  PROC DrawPart198()
    MoveL Offs(pOrigin,350.48,95.40,0.00),v40,z0,tPen\WObj:=wPaper;
    MoveL Offs(pOrigin,348.08,93.00,0.00),v40,z0,tPen\WObj:=wPaper;
    MoveL Offs(pOrigin,348.60,93.14,0.00),v40,z0,tPen\WObj:=wPaper;
    MoveL Offs(pOrigin,351.36,93.14,0.00),v40,z0,tPen\WObj:=wPaper;
    MoveL Offs(pOrigin,351.36,92.97,0.00),v40,z0,tPen\WObj:=wPaper;
    MoveL Offs(pOrigin,350.94,93.61,0.00),v40,z0,tPen\WObj:=wPaper;
    MoveL Offs(pOrigin,351.36,92.97,0.00),v40,z0,tPen\WObj:=wPaper;
    MoveL Offs(pOrigin,350.61,93.40,0.00),v40,z0,tPen\WObj:=wPaper;
    MoveL Offs(pOrigin,350.61,90.42,0.00),v40,z0,tPen\WObj:=wPaper;
    MoveL Offs(pOrigin,350.30,90.64,0.00),v40,z0,tPen\WObj:=wPaper;
    MoveL Offs(pOrigin,348.60,77.25,0.00),v40,z0,tPen\WObj:=wPaper;
    MoveL Offs(pOrigin,348.81,76.82,0.00),v40,z0,tPen\WObj:=wPaper;
    MoveL Offs(pOrigin,351.36,77.04,0.00),v40,z0,tPen\WObj:=wPaper;
    MoveL Offs(pOrigin,352.42,77.46,0.00),v40,z0,tPen\WObj:=wPaper;
    MoveL Offs(pOrigin,351.79,82.35,0.00),v40,z0,tPen\WObj:=wPaper;
    MoveL Offs(pOrigin,351.58,87.66,0.00),v40,z0,tPen\WObj:=wPaper;
    MoveL Offs(pOrigin,350.94,90.21,0.00),v40,z0,tPen\WObj:=wPaper;
    MoveL Offs(pOrigin,350.30,91.28,0.00),v40,fine,tPen\WObj:=wPaper;
    MoveL Offs(pOrigin,350.30,91.28,6.00),v60,z5,tPen\WObj:=wPaper;
    MoveL Offs(pOrigin,348.07,90.00,6.00),vTravel,z5,tPen\WObj:=wPaper;
    MoveL Offs(pOrigin,348.07,90.00,0.00),v60,z0,tPen\WObj:=wPaper;
    MoveL Offs(pOrigin,351.83,93.76,0.00),v40,z0,tPen\WObj:=wPaper;
    MoveL Offs(pOrigin,350.73,93.82,0.00),v40,z0,tPen\WObj:=wPaper;
    MoveL Offs(pOrigin,350.30,94.46,0.00),v40,z0,tPen\WObj:=wPaper;
    MoveL Offs(pOrigin,350.73,93.82,0.00),v40,fine,tPen\WObj:=wPaper;
    MoveL Offs(pOrigin,350.73,93.82,6.00),v60,z5,tPen\WObj:=wPaper;
    MoveL Offs(pOrigin,347.54,90.28,6.00),vTravel,z5,tPen\WObj:=wPaper;
    MoveL Offs(pOrigin,347.54,90.28,0.00),v60,z0,tPen\WObj:=wPaper;
    MoveL Offs(pOrigin,354.30,83.51,0.00),v40,z0,tPen\WObj:=wPaper;
    MoveL Offs(pOrigin,353.89,83.88,0.00),v40,z0,tPen\WObj:=wPaper;
    MoveL Offs(pOrigin,351.49,81.47,0.00),v40,z0,tPen\WObj:=wPaper;
    MoveL Offs(pOrigin,352.00,81.53,0.00),v40,z0,tPen\WObj:=wPaper;
    MoveL Offs(pOrigin,353.49,81.53,0.00),v40,z0,tPen\WObj:=wPaper;
    MoveL Offs(pOrigin,354.03,81.03,0.00),v40,z0,tPen\WObj:=wPaper;
    MoveL Offs(pOrigin,351.63,78.63,0.00),v40,z0,tPen\WObj:=wPaper;
    MoveL Offs(pOrigin,352.21,78.36,0.00),v40,z0,tPen\WObj:=wPaper;
    MoveL Offs(pOrigin,354.12,78.36,0.00),v40,z0,tPen\WObj:=wPaper;
    MoveL Offs(pOrigin,353.77,77.89,0.00),v40,z0,tPen\WObj:=wPaper;
    MoveL Offs(pOrigin,353.77,76.40,0.00),v40,fine,tPen\WObj:=wPaper;
    MoveL Offs(pOrigin,353.77,76.40,6.00),v60,z5,tPen\WObj:=wPaper;
    MoveL Offs(pOrigin,352.53,74.83,6.00),vTravel,z5,tPen\WObj:=wPaper;
    MoveL Offs(pOrigin,352.53,74.83,0.00),v60,z0,tPen\WObj:=wPaper;
    MoveL Offs(pOrigin,346.52,80.84,0.00),v40,fine,tPen\WObj:=wPaper;
    MoveL Offs(pOrigin,346.52,80.84,6.00),v60,z5,tPen\WObj:=wPaper;
    MoveL Offs(pOrigin,346.38,79.49,6.00),vTravel,z5,tPen\WObj:=wPaper;
    MoveL Offs(pOrigin,346.38,79.49,0.00),v60,z0,tPen\WObj:=wPaper;
    MoveL Offs(pOrigin,351.34,74.54,0.00),v40,z0,tPen\WObj:=wPaper;
    MoveL Offs(pOrigin,351.17,75.18,0.00),v40,z0,tPen\WObj:=wPaper;
    MoveL Offs(pOrigin,354.93,78.94,0.00),v40,fine,tPen\WObj:=wPaper;
    MoveL Offs(pOrigin,354.93,78.94,6.00),v60,z5,tPen\WObj:=wPaper;
    MoveL Offs(pOrigin,355.66,80.66,6.00),vTravel,z5,tPen\WObj:=wPaper;
    MoveL Offs(pOrigin,355.66,80.66,0.00),v60,z0,tPen\WObj:=wPaper;
    MoveL Offs(pOrigin,361.07,75.25,0.00),v40,z0,tPen\WObj:=wPaper;
    MoveL Offs(pOrigin,360.76,75.81,0.00),v40,z0,tPen\WObj:=wPaper;
    MoveL Offs(pOrigin,368.57,83.62,0.00),v40,z0,tPen\WObj:=wPaper;
    MoveL Offs(pOrigin,368.83,83.92,0.00),v40,z0,tPen\WObj:=wPaper;
    MoveL Offs(pOrigin,373.49,79.26,0.00),v40,z0,tPen\WObj:=wPaper;
    MoveL Offs(pOrigin,373.65,79.75,0.00),v40,z0,tPen\WObj:=wPaper;
    MoveL Offs(pOrigin,374.86,80.95,0.00),v40,fine,tPen\WObj:=wPaper;
    MoveL Offs(pOrigin,374.86,80.95,6.00),v60,z5,tPen\WObj:=wPaper;
    MoveL Offs(pOrigin,373.36,80.94,6.00),vTravel,z5,tPen\WObj:=wPaper;
    MoveL Offs(pOrigin,373.36,80.94,0.00),v60,z0,tPen\WObj:=wPaper;
    MoveL Offs(pOrigin,372.46,80.04,0.00),v40,z0,tPen\WObj:=wPaper;
    MoveL Offs(pOrigin,371.99,79.27,0.00),v40,z0,tPen\WObj:=wPaper;
    MoveL Offs(pOrigin,367.79,83.47,0.00),v40,z0,tPen\WObj:=wPaper;
    MoveL Offs(pOrigin,366.89,82.88,0.00),v40,z0,tPen\WObj:=wPaper;
    MoveL Offs(pOrigin,370.49,79.27,0.00),v40,z0,tPen\WObj:=wPaper;
    MoveL Offs(pOrigin,370.96,80.04,0.00),v40,z0,tPen\WObj:=wPaper;
    MoveL Offs(pOrigin,371.86,80.94,0.00),v40,fine,tPen\WObj:=wPaper;
    MoveL Offs(pOrigin,371.86,80.94,6.00),v60,z5,tPen\WObj:=wPaper;
    MoveL Offs(pOrigin,372.40,82.58,6.00),vTravel,z5,tPen\WObj:=wPaper;
    MoveL Offs(pOrigin,372.40,82.58,0.00),v60,z0,tPen\WObj:=wPaper;
    MoveL Offs(pOrigin,368.58,82.58,0.00),v40,fine,tPen\WObj:=wPaper;
    MoveL Offs(pOrigin,368.58,82.58,6.00),v60,z5,tPen\WObj:=wPaper;
    MoveL Offs(pOrigin,370.06,81.53,6.00),vTravel,z5,tPen\WObj:=wPaper;
    MoveL Offs(pOrigin,370.06,81.53,0.00),v60,z0,tPen\WObj:=wPaper;
    MoveL Offs(pOrigin,366.45,81.53,0.00),v40,fine,tPen\WObj:=wPaper;
    MoveL Offs(pOrigin,366.45,81.53,6.00),v60,z5,tPen\WObj:=wPaper;
    MoveL Offs(pOrigin,364.94,81.83,6.00),vTravel,z5,tPen\WObj:=wPaper;
    MoveL Offs(pOrigin,364.94,81.83,0.00),v60,z0,tPen\WObj:=wPaper;
    MoveL Offs(pOrigin,367.80,78.98,0.00),v40,fine,tPen\WObj:=wPaper;
    MoveL Offs(pOrigin,367.80,78.98,6.00),v60,z5,tPen\WObj:=wPaper;
    MoveL Offs(pOrigin,368.36,80.47,6.00),vTravel,z5,tPen\WObj:=wPaper;
    MoveL Offs(pOrigin,368.36,80.47,0.00),v60,z0,tPen\WObj:=wPaper;
    MoveL Offs(pOrigin,364.54,80.47,0.00),v40,fine,tPen\WObj:=wPaper;
    MoveL Offs(pOrigin,364.54,80.47,6.00),v60,z5,tPen\WObj:=wPaper;
    MoveL Offs(pOrigin,366.24,79.42,6.00),vTravel,z5,tPen\WObj:=wPaper;
    MoveL Offs(pOrigin,366.24,79.42,0.00),v60,z0,tPen\WObj:=wPaper;
    MoveL Offs(pOrigin,362.84,79.42,0.00),v40,z0,tPen\WObj:=wPaper;
    MoveL Offs(pOrigin,362.22,78.74,0.00),v40,z0,tPen\WObj:=wPaper;
    MoveL Offs(pOrigin,362.22,77.04,0.00),v40,z0,tPen\WObj:=wPaper;
    MoveL Offs(pOrigin,361.17,76.82,0.00),v40,z0,tPen\WObj:=wPaper;
    MoveL Offs(pOrigin,361.17,78.31,0.00),v40,fine,tPen\WObj:=wPaper;
    MoveL Offs(pOrigin,361.17,78.31,6.00),v60,z5,tPen\WObj:=wPaper;
    MoveL Offs(pOrigin,359.11,78.71,6.00),vTravel,z5,tPen\WObj:=wPaper;
    MoveL Offs(pOrigin,359.11,78.71,0.00),v60,z0,tPen\WObj:=wPaper;
    MoveL Offs(pOrigin,362.42,75.40,0.00),v40,fine,tPen\WObj:=wPaper;
    MoveL Offs(pOrigin,362.42,75.40,6.00),v60,z5,tPen\WObj:=wPaper;
    MoveL Offs(pOrigin,360.14,69.22,6.00),vTravel,z5,tPen\WObj:=wPaper;
    MoveL Offs(pOrigin,360.14,69.22,0.00),v60,z0,tPen\WObj:=wPaper;
    MoveL Offs(pOrigin,359.24,68.32,0.00),v40,fine,tPen\WObj:=wPaper;
    MoveL Offs(pOrigin,359.24,68.32,6.00),v60,z5,tPen\WObj:=wPaper;
    MoveL Offs(pOrigin,361.33,67.42,6.00),vTravel,z5,tPen\WObj:=wPaper;
    MoveL Offs(pOrigin,361.33,67.42,0.00),v60,z0,tPen\WObj:=wPaper;
    MoveL Offs(pOrigin,362.23,68.33,0.00),v40,z0,tPen\WObj:=wPaper;
    MoveL Offs(pOrigin,363.28,67.88,0.00),v40,z0,tPen\WObj:=wPaper;
    MoveL Offs(pOrigin,362.38,66.98,0.00),v40,fine,tPen\WObj:=wPaper;
    MoveL Offs(pOrigin,362.38,66.98,6.00),v60,z5,tPen\WObj:=wPaper;
    MoveL Offs(pOrigin,364.32,65.94,6.00),vTravel,z5,tPen\WObj:=wPaper;
    MoveL Offs(pOrigin,364.32,65.94,0.00),v60,z0,tPen\WObj:=wPaper;
    MoveL Offs(pOrigin,365.23,66.84,0.00),v40,z0,tPen\WObj:=wPaper;
    MoveL Offs(pOrigin,366.27,66.39,0.00),v40,z0,tPen\WObj:=wPaper;
    MoveL Offs(pOrigin,365.37,65.49,0.00),v40,fine,tPen\WObj:=wPaper;
    MoveL Offs(pOrigin,365.37,65.49,6.00),v60,z5,tPen\WObj:=wPaper;
    MoveL Offs(pOrigin,371.09,75.69,6.00),vTravel,z5,tPen\WObj:=wPaper;
    MoveL Offs(pOrigin,371.09,75.69,0.00),v60,z0,tPen\WObj:=wPaper;
    MoveL Offs(pOrigin,371.85,76.44,0.00),v40,fine,tPen\WObj:=wPaper;
    MoveL Offs(pOrigin,371.85,76.44,6.00),v60,z5,tPen\WObj:=wPaper;
    MoveL Offs(pOrigin,377.37,82.84,6.00),vTravel,z5,tPen\WObj:=wPaper;
    MoveL Offs(pOrigin,377.37,82.84,0.00),v60,z0,tPen\WObj:=wPaper;
  ENDPROC

  PROC DrawPart199()
    MoveL Offs(pOrigin,374.52,85.70,0.00),v40,fine,tPen\WObj:=wPaper;
    MoveL Offs(pOrigin,374.52,85.70,6.00),v60,z5,tPen\WObj:=wPaper;
    MoveL Offs(pOrigin,370.74,95.45,6.00),vTravel,z5,tPen\WObj:=wPaper;
    MoveL Offs(pOrigin,370.74,95.45,0.00),v60,z0,tPen\WObj:=wPaper;
    MoveL Offs(pOrigin,369.39,96.80,0.00),v40,z0,tPen\WObj:=wPaper;
    MoveL Offs(pOrigin,368.35,96.35,0.00),v40,z0,tPen\WObj:=wPaper;
    MoveL Offs(pOrigin,369.70,95.00,0.00),v40,z0,tPen\WObj:=wPaper;
    MoveL Offs(pOrigin,368.65,94.56,0.00),v40,z0,tPen\WObj:=wPaper;
    MoveL Offs(pOrigin,367.30,95.91,0.00),v40,fine,tPen\WObj:=wPaper;
    MoveL Offs(pOrigin,367.30,95.91,6.00),v60,z5,tPen\WObj:=wPaper;
    MoveL Offs(pOrigin,370.44,97.25,6.00),vTravel,z5,tPen\WObj:=wPaper;
    MoveL Offs(pOrigin,370.44,97.25,0.00),v60,z0,tPen\WObj:=wPaper;
    MoveL Offs(pOrigin,371.79,95.89,0.00),v40,z0,tPen\WObj:=wPaper;
    MoveL Offs(pOrigin,372.84,96.34,0.00),v40,z0,tPen\WObj:=wPaper;
    MoveL Offs(pOrigin,371.79,97.39,0.00),v40,fine,tPen\WObj:=wPaper;
    MoveL Offs(pOrigin,371.79,97.39,6.00),v60,z5,tPen\WObj:=wPaper;
    MoveL Offs(pOrigin,373.14,97.54,6.00),vTravel,z5,tPen\WObj:=wPaper;
    MoveL Offs(pOrigin,373.14,97.54,0.00),v60,z0,tPen\WObj:=wPaper;
    MoveL Offs(pOrigin,373.89,96.79,0.00),v40,fine,tPen\WObj:=wPaper;
    MoveL Offs(pOrigin,373.89,96.79,6.00),v60,z5,tPen\WObj:=wPaper;
    MoveL Offs(pOrigin,376.01,97.86,6.00),vTravel,z5,tPen\WObj:=wPaper;
    MoveL Offs(pOrigin,376.01,97.86,0.00),v60,z0,tPen\WObj:=wPaper;
    MoveL Offs(pOrigin,369.21,95.88,0.00),v40,z0,tPen\WObj:=wPaper;
    MoveL Offs(pOrigin,364.75,93.40,0.00),v40,z0,tPen\WObj:=wPaper;
    MoveL Offs(pOrigin,360.08,89.15,0.00),v40,z0,tPen\WObj:=wPaper;
    MoveL Offs(pOrigin,357.10,84.90,0.00),v40,fine,tPen\WObj:=wPaper;
    MoveL Offs(pOrigin,357.10,84.90,6.00),v60,z5,tPen\WObj:=wPaper;
    MoveL Offs(pOrigin,353.99,86.81,6.00),vTravel,z5,tPen\WObj:=wPaper;
    MoveL Offs(pOrigin,353.99,86.81,0.00),v60,z0,tPen\WObj:=wPaper;
    MoveL Offs(pOrigin,342.72,98.08,0.00),v40,fine,tPen\WObj:=wPaper;
    MoveL Offs(pOrigin,342.72,98.08,6.00),v60,z5,tPen\WObj:=wPaper;
    MoveL Offs(pOrigin,343.60,98.98,6.00),vTravel,z5,tPen\WObj:=wPaper;
    MoveL Offs(pOrigin,343.60,98.98,0.00),v60,z0,tPen\WObj:=wPaper;
    MoveL Offs(pOrigin,352.17,107.54,0.00),v40,z0,tPen\WObj:=wPaper;
    MoveL Offs(pOrigin,351.79,107.85,0.00),v40,z0,tPen\WObj:=wPaper;
    MoveL Offs(pOrigin,353.27,109.34,0.00),v40,z0,tPen\WObj:=wPaper;
    MoveL Offs(pOrigin,351.79,107.85,0.00),v40,fine,tPen\WObj:=wPaper;
    MoveL Offs(pOrigin,351.79,107.85,6.00),v60,z5,tPen\WObj:=wPaper;
    MoveL Offs(pOrigin,355.87,108.83,6.00),vTravel,z5,tPen\WObj:=wPaper;
    MoveL Offs(pOrigin,355.87,108.83,0.00),v60,z0,tPen\WObj:=wPaper;
    MoveL Offs(pOrigin,357.83,106.87,0.00),v40,z0,tPen\WObj:=wPaper;
    MoveL Offs(pOrigin,358.72,107.47,0.00),v40,z0,tPen\WObj:=wPaper;
    MoveL Offs(pOrigin,356.62,109.57,0.00),v40,z0,tPen\WObj:=wPaper;
    MoveL Offs(pOrigin,356.37,108.75,0.00),v40,z0,tPen\WObj:=wPaper;
    MoveL Offs(pOrigin,341.94,94.33,0.00),v40,z0,tPen\WObj:=wPaper;
    MoveL Offs(pOrigin,341.54,94.79,0.00),v40,z0,tPen\WObj:=wPaper;
    MoveL Offs(pOrigin,345.74,90.58,0.00),v40,z0,tPen\WObj:=wPaper;
    MoveL Offs(pOrigin,346.19,91.63,0.00),v40,z0,tPen\WObj:=wPaper;
    MoveL Offs(pOrigin,341.83,95.99,0.00),v40,fine,tPen\WObj:=wPaper;
    MoveL Offs(pOrigin,341.83,95.99,6.00),v60,z5,tPen\WObj:=wPaper;
    MoveL Offs(pOrigin,344.14,98.42,6.00),vTravel,z5,tPen\WObj:=wPaper;
    MoveL Offs(pOrigin,344.14,98.42,0.00),v60,z0,tPen\WObj:=wPaper;
    MoveL Offs(pOrigin,349.02,98.42,0.00),v40,fine,tPen\WObj:=wPaper;
    MoveL Offs(pOrigin,349.02,98.42,6.00),v60,z5,tPen\WObj:=wPaper;
    MoveL Offs(pOrigin,347.40,88.93,6.00),vTravel,z5,tPen\WObj:=wPaper;
    MoveL Offs(pOrigin,347.40,88.93,0.00),v60,z0,tPen\WObj:=wPaper;
    MoveL Offs(pOrigin,354.31,82.02,0.00),v40,fine,tPen\WObj:=wPaper;
    MoveL Offs(pOrigin,354.31,82.02,6.00),v60,z5,tPen\WObj:=wPaper;
    MoveL Offs(pOrigin,353.70,80.47,6.00),vTravel,z5,tPen\WObj:=wPaper;
    MoveL Offs(pOrigin,353.70,80.47,0.00),v60,z0,tPen\WObj:=wPaper;
    MoveL Offs(pOrigin,352.00,80.47,0.00),v40,fine,tPen\WObj:=wPaper;
    MoveL Offs(pOrigin,352.00,80.47,6.00),v60,z5,tPen\WObj:=wPaper;
    MoveL Offs(pOrigin,351.17,79.18,6.00),vTravel,z5,tPen\WObj:=wPaper;
    MoveL Offs(pOrigin,351.17,79.18,0.00),v60,z0,tPen\WObj:=wPaper;
    MoveL Offs(pOrigin,355.38,74.97,0.00),v40,fine,tPen\WObj:=wPaper;
    MoveL Offs(pOrigin,355.38,74.97,6.00),v60,z5,tPen\WObj:=wPaper;
    MoveL Offs(pOrigin,350.58,77.58,6.00),vTravel,z5,tPen\WObj:=wPaper;
    MoveL Offs(pOrigin,350.58,77.58,0.00),v60,z0,tPen\WObj:=wPaper;
    MoveL Offs(pOrigin,347.72,74.72,0.00),v40,z0,tPen\WObj:=wPaper;
    MoveL Offs(pOrigin,347.44,75.55,0.00),v40,z0,tPen\WObj:=wPaper;
    MoveL Offs(pOrigin,347.44,77.68,0.00),v40,z0,tPen\WObj:=wPaper;
    MoveL Offs(pOrigin,347.11,77.30,0.00),v40,z0,tPen\WObj:=wPaper;
    MoveL Offs(pOrigin,349.02,77.30,0.00),v40,z0,tPen\WObj:=wPaper;
    MoveL Offs(pOrigin,348.49,77.04,0.00),v40,z0,tPen\WObj:=wPaper;
    MoveL Offs(pOrigin,348.49,75.76,0.00),v40,z0,tPen\WObj:=wPaper;
    MoveL Offs(pOrigin,349.45,75.19,0.00),v40,z0,tPen\WObj:=wPaper;
    MoveL Offs(pOrigin,337.34,75.19,0.00),v40,z0,tPen\WObj:=wPaper;
    MoveL Offs(pOrigin,337.98,75.76,0.00),v40,z0,tPen\WObj:=wPaper;
    MoveL Offs(pOrigin,336.06,74.91,0.00),v40,z0,tPen\WObj:=wPaper;
    MoveL Offs(pOrigin,334.58,74.70,0.00),v40,z0,tPen\WObj:=wPaper;
    MoveL Offs(pOrigin,334.15,74.91,0.00),v40,z0,tPen\WObj:=wPaper;
    MoveL Offs(pOrigin,333.65,75.79,0.00),v40,z0,tPen\WObj:=wPaper;
    MoveL Offs(pOrigin,336.66,72.78,0.00),v40,fine,tPen\WObj:=wPaper;
    MoveL Offs(pOrigin,336.66,72.78,6.00),v60,z5,tPen\WObj:=wPaper;
    MoveL Offs(pOrigin,346.07,74.57,6.00),vTravel,z5,tPen\WObj:=wPaper;
    MoveL Offs(pOrigin,346.07,74.57,0.00),v60,z0,tPen\WObj:=wPaper;
    MoveL Offs(pOrigin,349.38,77.87,0.00),v40,z0,tPen\WObj:=wPaper;
    MoveL Offs(pOrigin,348.81,78.36,0.00),v40,z0,tPen\WObj:=wPaper;
    MoveL Offs(pOrigin,347.33,78.36,0.00),v40,fine,tPen\WObj:=wPaper;
    MoveL Offs(pOrigin,347.33,78.36,6.00),v60,z5,tPen\WObj:=wPaper;
    MoveL Offs(pOrigin,351.79,83.64,6.00),vTravel,z5,tPen\WObj:=wPaper;
    MoveL Offs(pOrigin,351.79,83.64,0.00),v60,z0,tPen\WObj:=wPaper;
    MoveL Offs(pOrigin,353.28,83.64,0.00),v40,fine,tPen\WObj:=wPaper;
    MoveL Offs(pOrigin,353.28,83.64,6.00),v60,z5,tPen\WObj:=wPaper;
    MoveL Offs(pOrigin,353.28,85.75,6.00),vTravel,z5,tPen\WObj:=wPaper;
    MoveL Offs(pOrigin,353.28,85.75,0.00),v60,z0,tPen\WObj:=wPaper;
    MoveL Offs(pOrigin,351.58,85.75,0.00),v40,fine,tPen\WObj:=wPaper;
    MoveL Offs(pOrigin,351.58,85.75,6.00),v60,z5,tPen\WObj:=wPaper;
    MoveL Offs(pOrigin,344.85,88.49,6.00),vTravel,z5,tPen\WObj:=wPaper;
    MoveL Offs(pOrigin,344.85,88.49,0.00),v60,z0,tPen\WObj:=wPaper;
    MoveL Offs(pOrigin,340.64,92.69,0.00),v40,fine,tPen\WObj:=wPaper;
    MoveL Offs(pOrigin,340.64,92.69,6.00),v60,z5,tPen\WObj:=wPaper;
    MoveL Offs(pOrigin,344.17,87.59,6.00),vTravel,z5,tPen\WObj:=wPaper;
    MoveL Offs(pOrigin,344.17,87.59,0.00),v60,z0,tPen\WObj:=wPaper;
    MoveL Offs(pOrigin,340.86,84.29,0.00),v40,fine,tPen\WObj:=wPaper;
    MoveL Offs(pOrigin,340.86,84.29,6.00),v60,z5,tPen\WObj:=wPaper;
    MoveL Offs(pOrigin,338.19,83.41,6.00),vTravel,z5,tPen\WObj:=wPaper;
    MoveL Offs(pOrigin,338.19,83.41,0.00),v60,z0,tPen\WObj:=wPaper;
    MoveL Offs(pOrigin,338.40,83.84,0.00),v40,z0,tPen\WObj:=wPaper;
    MoveL Offs(pOrigin,338.19,83.41,0.00),v40,fine,tPen\WObj:=wPaper;
    MoveL Offs(pOrigin,338.19,83.41,6.00),v60,z5,tPen\WObj:=wPaper;
    MoveL Offs(pOrigin,325.28,70.72,6.00),vTravel,z5,tPen\WObj:=wPaper;
    MoveL Offs(pOrigin,325.28,70.72,0.00),v60,z0,tPen\WObj:=wPaper;
    MoveL Offs(pOrigin,322.73,73.28,0.00),v40,fine,tPen\WObj:=wPaper;
    MoveL Offs(pOrigin,322.73,73.28,6.00),v60,z5,tPen\WObj:=wPaper;
    MoveL Offs(pOrigin,327.93,66.87,6.00),vTravel,z5,tPen\WObj:=wPaper;
    MoveL Offs(pOrigin,327.93,66.87,0.00),v60,z0,tPen\WObj:=wPaper;
    MoveL Offs(pOrigin,326.42,65.37,0.00),v40,fine,tPen\WObj:=wPaper;
    MoveL Offs(pOrigin,326.42,65.37,6.00),v60,z5,tPen\WObj:=wPaper;
    MoveL Offs(pOrigin,294.88,66.77,6.00),vTravel,z5,tPen\WObj:=wPaper;
  ENDPROC

  PROC DrawPart200()
    MoveL Offs(pOrigin,294.88,66.77,0.00),v60,z0,tPen\WObj:=wPaper;
    MoveL Offs(pOrigin,292.63,69.02,0.00),v40,fine,tPen\WObj:=wPaper;
    MoveL Offs(pOrigin,292.63,69.02,6.00),v60,z5,tPen\WObj:=wPaper;
    MoveL Offs(pOrigin,292.18,70.97,6.00),vTravel,z5,tPen\WObj:=wPaper;
    MoveL Offs(pOrigin,292.18,70.97,0.00),v60,z0,tPen\WObj:=wPaper;
    MoveL Offs(pOrigin,294.58,68.57,0.00),v40,fine,tPen\WObj:=wPaper;
    MoveL Offs(pOrigin,294.58,68.57,6.00),v60,z5,tPen\WObj:=wPaper;
    MoveL Offs(pOrigin,294.42,70.22,6.00),vTravel,z5,tPen\WObj:=wPaper;
    MoveL Offs(pOrigin,294.42,70.22,0.00),v60,z0,tPen\WObj:=wPaper;
    MoveL Offs(pOrigin,291.72,72.92,0.00),v40,fine,tPen\WObj:=wPaper;
    MoveL Offs(pOrigin,291.72,72.92,6.00),v60,z5,tPen\WObj:=wPaper;
    MoveL Offs(pOrigin,291.57,74.57,6.00),vTravel,z5,tPen\WObj:=wPaper;
    MoveL Offs(pOrigin,291.57,74.57,0.00),v60,z0,tPen\WObj:=wPaper;
    MoveL Offs(pOrigin,293.97,72.17,0.00),v40,fine,tPen\WObj:=wPaper;
    MoveL Offs(pOrigin,293.97,72.17,6.00),v60,z5,tPen\WObj:=wPaper;
    MoveL Offs(pOrigin,293.81,73.81,6.00),vTravel,z5,tPen\WObj:=wPaper;
    MoveL Offs(pOrigin,293.81,73.81,0.00),v60,z0,tPen\WObj:=wPaper;
    MoveL Offs(pOrigin,291.41,76.22,0.00),v40,fine,tPen\WObj:=wPaper;
    MoveL Offs(pOrigin,291.41,76.22,6.00),v60,z5,tPen\WObj:=wPaper;
    MoveL Offs(pOrigin,291.11,78.02,6.00),vTravel,z5,tPen\WObj:=wPaper;
    MoveL Offs(pOrigin,291.11,78.02,0.00),v60,z0,tPen\WObj:=wPaper;
    MoveL Offs(pOrigin,293.51,75.61,0.00),v40,fine,tPen\WObj:=wPaper;
    MoveL Offs(pOrigin,293.51,75.61,6.00),v60,z5,tPen\WObj:=wPaper;
    MoveL Offs(pOrigin,287.97,73.68,6.00),vTravel,z5,tPen\WObj:=wPaper;
    MoveL Offs(pOrigin,287.97,73.68,0.00),v60,z0,tPen\WObj:=wPaper;
    MoveL Offs(pOrigin,285.27,76.39,0.00),v40,fine,tPen\WObj:=wPaper;
    MoveL Offs(pOrigin,285.27,76.39,6.00),v60,z5,tPen\WObj:=wPaper;
    MoveL Offs(pOrigin,288.98,66.75,6.00),vTravel,z5,tPen\WObj:=wPaper;
    MoveL Offs(pOrigin,288.98,66.75,0.00),v60,z0,tPen\WObj:=wPaper;
    MoveL Offs(pOrigin,287.47,65.25,0.00),v40,z0,tPen\WObj:=wPaper;
    MoveL Offs(pOrigin,287.61,65.69,0.00),v40,z0,tPen\WObj:=wPaper;
    MoveL Offs(pOrigin,289.74,65.69,0.00),v40,fine,tPen\WObj:=wPaper;
    MoveL Offs(pOrigin,289.74,65.69,6.00),v60,z5,tPen\WObj:=wPaper;
    MoveL Offs(pOrigin,280.60,66.74,6.00),vTravel,z5,tPen\WObj:=wPaper;
    MoveL Offs(pOrigin,280.60,66.74,0.00),v60,z0,tPen\WObj:=wPaper;
    MoveL Offs(pOrigin,274.44,66.74,0.00),v40,z0,tPen\WObj:=wPaper;
    MoveL Offs(pOrigin,274.57,66.20,0.00),v40,z0,tPen\WObj:=wPaper;
    MoveL Offs(pOrigin,274.57,64.92,0.00),v40,z0,tPen\WObj:=wPaper;
    MoveL Offs(pOrigin,274.23,65.69,0.00),v40,z0,tPen\WObj:=wPaper;
    MoveL Offs(pOrigin,277.62,65.69,0.00),v40,z0,tPen\WObj:=wPaper;
    MoveL Offs(pOrigin,277.66,64.58,0.00),v40,z0,tPen\WObj:=wPaper;
    MoveL Offs(pOrigin,272.56,69.68,0.00),v40,fine,tPen\WObj:=wPaper;
    MoveL Offs(pOrigin,272.56,69.68,6.00),v60,z5,tPen\WObj:=wPaper;
    MoveL Offs(pOrigin,274.01,68.86,6.00),vTravel,z5,tPen\WObj:=wPaper;
    MoveL Offs(pOrigin,274.01,68.86,0.00),v60,z0,tPen\WObj:=wPaper;
    MoveL Offs(pOrigin,275.29,68.86,0.00),v40,z0,tPen\WObj:=wPaper;
    MoveL Offs(pOrigin,274.57,69.18,0.00),v40,z0,tPen\WObj:=wPaper;
    MoveL Offs(pOrigin,274.57,70.45,0.00),v40,fine,tPen\WObj:=wPaper;
    MoveL Offs(pOrigin,274.57,70.45,6.00),v60,z5,tPen\WObj:=wPaper;
    MoveL Offs(pOrigin,274.23,67.80,6.00),vTravel,z5,tPen\WObj:=wPaper;
    MoveL Offs(pOrigin,274.23,67.80,0.00),v60,z0,tPen\WObj:=wPaper;
    MoveL Offs(pOrigin,275.50,67.80,0.00),v40,z0,tPen\WObj:=wPaper;
    MoveL Offs(pOrigin,275.63,66.84,0.00),v40,z0,tPen\WObj:=wPaper;
    MoveL Offs(pOrigin,275.63,65.14,0.00),v40,fine,tPen\WObj:=wPaper;
    MoveL Offs(pOrigin,275.63,65.14,6.00),v60,z5,tPen\WObj:=wPaper;
    MoveL Offs(pOrigin,274.67,63.09,6.00),vTravel,z5,tPen\WObj:=wPaper;
    MoveL Offs(pOrigin,274.67,63.09,0.00),v60,z0,tPen\WObj:=wPaper;
    MoveL Offs(pOrigin,272.12,65.64,0.00),v40,z0,tPen\WObj:=wPaper;
    MoveL Offs(pOrigin,271.22,65.04,0.00),v40,z0,tPen\WObj:=wPaper;
    MoveL Offs(pOrigin,273.63,62.64,0.00),v40,z0,tPen\WObj:=wPaper;
    MoveL Offs(pOrigin,272.73,62.04,0.00),v40,z0,tPen\WObj:=wPaper;
    MoveL Offs(pOrigin,270.17,64.60,0.00),v40,fine,tPen\WObj:=wPaper;
    MoveL Offs(pOrigin,270.17,64.60,6.00),v60,z5,tPen\WObj:=wPaper;
    MoveL Offs(pOrigin,267.93,63.86,6.00),vTravel,z5,tPen\WObj:=wPaper;
    MoveL Offs(pOrigin,267.93,63.86,0.00),v60,z0,tPen\WObj:=wPaper;
    MoveL Offs(pOrigin,277.10,54.69,0.00),v40,z0,tPen\WObj:=wPaper;
    MoveL Offs(pOrigin,276.05,54.24,0.00),v40,z0,tPen\WObj:=wPaper;
    MoveL Offs(pOrigin,266.88,63.41,0.00),v40,z0,tPen\WObj:=wPaper;
    MoveL Offs(pOrigin,265.84,62.96,0.00),v40,z0,tPen\WObj:=wPaper;
    MoveL Offs(pOrigin,274.85,53.95,0.00),v40,z0,tPen\WObj:=wPaper;
    MoveL Offs(pOrigin,275.46,54.73,0.00),v40,z0,tPen\WObj:=wPaper;
    MoveL Offs(pOrigin,278.61,57.88,0.00),v40,z0,tPen\WObj:=wPaper;
    MoveL Offs(pOrigin,278.28,57.98,0.00),v40,z0,tPen\WObj:=wPaper;
    MoveL Offs(pOrigin,280.09,56.18,0.00),v40,z0,tPen\WObj:=wPaper;
    MoveL Offs(pOrigin,279.19,55.58,0.00),v40,z0,tPen\WObj:=wPaper;
    MoveL Offs(pOrigin,277.09,57.69,0.00),v40,fine,tPen\WObj:=wPaper;
    MoveL Offs(pOrigin,277.09,57.69,6.00),v60,z5,tPen\WObj:=wPaper;
    MoveL Offs(pOrigin,279.18,58.58,6.00),vTravel,z5,tPen\WObj:=wPaper;
    MoveL Offs(pOrigin,279.18,58.58,0.00),v60,z0,tPen\WObj:=wPaper;
    MoveL Offs(pOrigin,280.98,56.78,0.00),v40,fine,tPen\WObj:=wPaper;
    MoveL Offs(pOrigin,280.98,56.78,6.00),v60,z5,tPen\WObj:=wPaper;
    MoveL Offs(pOrigin,279.96,57.70,6.00),vTravel,z5,tPen\WObj:=wPaper;
    MoveL Offs(pOrigin,279.96,57.70,0.00),v60,z0,tPen\WObj:=wPaper;
    MoveL Offs(pOrigin,274.86,56.00,0.00),v40,z0,tPen\WObj:=wPaper;
    MoveL Offs(pOrigin,274.37,56.21,0.00),v40,z0,tPen\WObj:=wPaper;
    MoveL Offs(pOrigin,274.01,57.06,0.00),v40,z0,tPen\WObj:=wPaper;
    MoveL Offs(pOrigin,272.95,57.49,0.00),v40,fine,tPen\WObj:=wPaper;
    MoveL Offs(pOrigin,272.95,57.49,6.00),v60,z5,tPen\WObj:=wPaper;
    MoveL Offs(pOrigin,272.74,56.18,6.00),vTravel,z5,tPen\WObj:=wPaper;
    MoveL Offs(pOrigin,272.74,56.18,0.00),v60,z0,tPen\WObj:=wPaper;
    MoveL Offs(pOrigin,274.86,56.18,0.00),v40,z0,tPen\WObj:=wPaper;
    MoveL Offs(pOrigin,274.72,56.97,0.00),v40,z0,tPen\WObj:=wPaper;
    MoveL Offs(pOrigin,270.81,53.07,0.00),v40,z0,tPen\WObj:=wPaper;
    MoveL Offs(pOrigin,270.51,52.31,0.00),v40,z0,tPen\WObj:=wPaper;
    MoveL Offs(pOrigin,268.11,54.72,0.00),v40,z0,tPen\WObj:=wPaper;
    MoveL Offs(pOrigin,267.21,54.12,0.00),v40,z0,tPen\WObj:=wPaper;
    MoveL Offs(pOrigin,269.46,51.87,0.00),v40,fine,tPen\WObj:=wPaper;
    MoveL Offs(pOrigin,269.46,51.87,6.00),v60,z5,tPen\WObj:=wPaper;
    MoveL Offs(pOrigin,271.56,52.76,6.00),vTravel,z5,tPen\WObj:=wPaper;
    MoveL Offs(pOrigin,271.56,52.76,0.00),v60,z0,tPen\WObj:=wPaper;
    MoveL Offs(pOrigin,268.55,55.77,0.00),v40,fine,tPen\WObj:=wPaper;
    MoveL Offs(pOrigin,268.55,55.77,6.00),v60,z5,tPen\WObj:=wPaper;
    MoveL Offs(pOrigin,269.98,55.13,6.00),vTravel,z5,tPen\WObj:=wPaper;
    MoveL Offs(pOrigin,269.98,55.13,0.00),v60,z0,tPen\WObj:=wPaper;
    MoveL Offs(pOrigin,275.08,55.13,0.00),v40,fine,tPen\WObj:=wPaper;
    MoveL Offs(pOrigin,275.08,55.13,6.00),v60,z5,tPen\WObj:=wPaper;
    MoveL Offs(pOrigin,272.74,55.36,6.00),vTravel,z5,tPen\WObj:=wPaper;
    MoveL Offs(pOrigin,272.74,55.36,0.00),v60,z0,tPen\WObj:=wPaper;
    MoveL Offs(pOrigin,272.95,55.79,0.00),v40,z0,tPen\WObj:=wPaper;
    MoveL Offs(pOrigin,272.74,55.36,0.00),v40,fine,tPen\WObj:=wPaper;
    MoveL Offs(pOrigin,272.74,55.36,6.00),v60,z5,tPen\WObj:=wPaper;
    MoveL Offs(pOrigin,265.30,71.51,6.00),vTravel,z5,tPen\WObj:=wPaper;
    MoveL Offs(pOrigin,265.30,71.51,0.00),v60,z0,tPen\WObj:=wPaper;
    MoveL Offs(pOrigin,265.94,72.15,0.00),v40,z0,tPen\WObj:=wPaper;
    MoveL Offs(pOrigin,265.30,71.51,0.00),v40,z0,tPen\WObj:=wPaper;
    MoveL Offs(pOrigin,265.92,72.07,0.00),v40,z0,tPen\WObj:=wPaper;
    MoveL Offs(pOrigin,269.38,75.53,0.00),v40,z0,tPen\WObj:=wPaper;
    MoveL Offs(pOrigin,269.12,75.97,0.00),v40,z0,tPen\WObj:=wPaper;
    MoveL Offs(pOrigin,269.55,76.61,0.00),v40,z0,tPen\WObj:=wPaper;
    MoveL Offs(pOrigin,269.12,75.97,0.00),v40,z0,tPen\WObj:=wPaper;
  ENDPROC

  PROC DrawPart201()
    MoveL Offs(pOrigin,269.76,76.82,0.00),v40,z0,tPen\WObj:=wPaper;
    MoveL Offs(pOrigin,270.19,77.46,0.00),v40,z0,tPen\WObj:=wPaper;
    MoveL Offs(pOrigin,269.76,76.82,0.00),v40,fine,tPen\WObj:=wPaper;
    MoveL Offs(pOrigin,269.76,76.82,6.00),v60,z5,tPen\WObj:=wPaper;
    MoveL Offs(pOrigin,268.94,77.78,6.00),vTravel,z5,tPen\WObj:=wPaper;
    MoveL Offs(pOrigin,268.94,77.78,0.00),v60,z0,tPen\WObj:=wPaper;
    MoveL Offs(pOrigin,270.74,75.98,0.00),v40,z0,tPen\WObj:=wPaper;
    MoveL Offs(pOrigin,269.99,75.23,0.00),v40,z0,tPen\WObj:=wPaper;
    MoveL Offs(pOrigin,268.34,76.89,0.00),v40,z0,tPen\WObj:=wPaper;
    MoveL Offs(pOrigin,267.59,77.64,0.00),v40,z0,tPen\WObj:=wPaper;
    MoveL Offs(pOrigin,266.54,78.69,0.00),v40,z0,tPen\WObj:=wPaper;
    MoveL Offs(pOrigin,265.79,77.94,0.00),v40,z0,tPen\WObj:=wPaper;
    MoveL Offs(pOrigin,266.84,76.89,0.00),v40,fine,tPen\WObj:=wPaper;
    MoveL Offs(pOrigin,266.84,76.89,6.00),v60,z5,tPen\WObj:=wPaper;
    MoveL Offs(pOrigin,267.85,74.49,6.00),vTravel,z5,tPen\WObj:=wPaper;
    MoveL Offs(pOrigin,267.85,74.49,0.00),v60,z0,tPen\WObj:=wPaper;
    MoveL Offs(pOrigin,268.49,75.12,0.00),v40,z0,tPen\WObj:=wPaper;
    MoveL Offs(pOrigin,267.85,74.49,0.00),v40,fine,tPen\WObj:=wPaper;
    MoveL Offs(pOrigin,267.85,74.49,6.00),v60,z5,tPen\WObj:=wPaper;
    MoveL Offs(pOrigin,266.58,73.00,6.00),vTravel,z5,tPen\WObj:=wPaper;
    MoveL Offs(pOrigin,266.58,73.00,0.00),v60,z0,tPen\WObj:=wPaper;
    MoveL Offs(pOrigin,267.42,73.85,0.00),v40,z0,tPen\WObj:=wPaper;
    MoveL Offs(pOrigin,266.58,73.00,0.00),v40,fine,tPen\WObj:=wPaper;
    MoveL Offs(pOrigin,266.58,73.00,6.00),v60,z5,tPen\WObj:=wPaper;
    MoveL Offs(pOrigin,261.26,71.09,6.00),vTravel,z5,tPen\WObj:=wPaper;
    MoveL Offs(pOrigin,261.26,71.09,0.00),v60,z0,tPen\WObj:=wPaper;
    MoveL Offs(pOrigin,265.73,76.40,0.00),v40,z0,tPen\WObj:=wPaper;
    MoveL Offs(pOrigin,269.34,81.93,0.00),v40,fine,tPen\WObj:=wPaper;
    MoveL Offs(pOrigin,269.34,81.93,6.00),v60,z5,tPen\WObj:=wPaper;
    MoveL Offs(pOrigin,272.10,82.58,6.00),vTravel,z5,tPen\WObj:=wPaper;
    MoveL Offs(pOrigin,272.10,82.58,0.00),v60,z0,tPen\WObj:=wPaper;
    MoveL Offs(pOrigin,273.16,82.58,0.00),v40,fine,tPen\WObj:=wPaper;
    MoveL Offs(pOrigin,273.16,82.58,6.00),v60,z5,tPen\WObj:=wPaper;
    MoveL Offs(pOrigin,274.47,81.21,6.00),vTravel,z5,tPen\WObj:=wPaper;
    MoveL Offs(pOrigin,274.47,81.21,0.00),v60,z0,tPen\WObj:=wPaper;
    MoveL Offs(pOrigin,270.56,85.12,0.00),v40,z0,tPen\WObj:=wPaper;
    MoveL Offs(pOrigin,271.68,84.70,0.00),v40,z0,tPen\WObj:=wPaper;
    MoveL Offs(pOrigin,272.95,84.70,0.00),v40,z0,tPen\WObj:=wPaper;
    MoveL Offs(pOrigin,274.01,84.66,0.00),v40,z0,tPen\WObj:=wPaper;
    MoveL Offs(pOrigin,270.40,88.27,0.00),v40,z0,tPen\WObj:=wPaper;
    MoveL Offs(pOrigin,270.62,88.72,0.00),v40,z0,tPen\WObj:=wPaper;
    MoveL Offs(pOrigin,272.87,90.97,0.00),v40,z0,tPen\WObj:=wPaper;
    MoveL Offs(pOrigin,272.31,91.03,0.00),v40,z0,tPen\WObj:=wPaper;
    MoveL Offs(pOrigin,271.25,91.03,0.00),v40,z0,tPen\WObj:=wPaper;
    MoveL Offs(pOrigin,271.25,89.98,0.00),v40,z0,tPen\WObj:=wPaper;
    MoveL Offs(pOrigin,272.52,89.98,0.00),v40,z0,tPen\WObj:=wPaper;
    MoveL Offs(pOrigin,272.52,88.92,0.00),v40,z0,tPen\WObj:=wPaper;
    MoveL Offs(pOrigin,271.46,88.92,0.00),v40,fine,tPen\WObj:=wPaper;
    MoveL Offs(pOrigin,271.46,88.92,6.00),v60,z5,tPen\WObj:=wPaper;
    MoveL Offs(pOrigin,273.39,91.25,6.00),vTravel,z5,tPen\WObj:=wPaper;
    MoveL Offs(pOrigin,273.39,91.25,0.00),v60,z0,tPen\WObj:=wPaper;
    MoveL Offs(pOrigin,269.63,95.01,0.00),v40,fine,tPen\WObj:=wPaper;
    MoveL Offs(pOrigin,269.63,95.01,6.00),v60,z5,tPen\WObj:=wPaper;
    MoveL Offs(pOrigin,270.83,78.53,6.00),vTravel,z5,tPen\WObj:=wPaper;
    MoveL Offs(pOrigin,270.83,78.53,0.00),v60,z0,tPen\WObj:=wPaper;
    MoveL Offs(pOrigin,271.04,78.95,0.00),v40,z0,tPen\WObj:=wPaper;
    MoveL Offs(pOrigin,270.83,78.53,0.00),v40,fine,tPen\WObj:=wPaper;
    MoveL Offs(pOrigin,270.83,78.53,6.00),v60,z5,tPen\WObj:=wPaper;
    MoveL Offs(pOrigin,288.25,86.81,6.00),vTravel,z5,tPen\WObj:=wPaper;
    MoveL Offs(pOrigin,288.25,86.81,0.00),v60,z0,tPen\WObj:=wPaper;
    MoveL Offs(pOrigin,289.52,86.81,0.00),v40,fine,tPen\WObj:=wPaper;
    MoveL Offs(pOrigin,289.52,86.81,6.00),v60,z5,tPen\WObj:=wPaper;
    MoveL Offs(pOrigin,293.02,88.05,6.00),vTravel,z5,tPen\WObj:=wPaper;
    MoveL Offs(pOrigin,293.02,88.05,0.00),v60,z0,tPen\WObj:=wPaper;
    MoveL Offs(pOrigin,288.51,92.55,0.00),v40,fine,tPen\WObj:=wPaper;
    MoveL Offs(pOrigin,288.51,92.55,6.00),v60,z5,tPen\WObj:=wPaper;
    MoveL Offs(pOrigin,288.81,93.75,6.00),vTravel,z5,tPen\WObj:=wPaper;
    MoveL Offs(pOrigin,288.81,93.75,0.00),v60,z0,tPen\WObj:=wPaper;
    MoveL Offs(pOrigin,293.02,89.54,0.00),v40,fine,tPen\WObj:=wPaper;
    MoveL Offs(pOrigin,293.02,89.54,6.00),v60,z5,tPen\WObj:=wPaper;
    MoveL Offs(pOrigin,292.92,99.48,6.00),vTravel,z5,tPen\WObj:=wPaper;
    MoveL Offs(pOrigin,292.92,99.48,0.00),v60,z0,tPen\WObj:=wPaper;
    MoveL Offs(pOrigin,291.44,99.48,0.00),v40,fine,tPen\WObj:=wPaper;
    MoveL Offs(pOrigin,291.44,99.48,6.00),v60,z5,tPen\WObj:=wPaper;
    MoveL Offs(pOrigin,293.88,100.63,6.00),vTravel,z5,tPen\WObj:=wPaper;
    MoveL Offs(pOrigin,293.88,100.63,0.00),v60,z0,tPen\WObj:=wPaper;
    MoveL Offs(pOrigin,291.33,103.18,0.00),v40,fine,tPen\WObj:=wPaper;
    MoveL Offs(pOrigin,291.33,103.18,6.00),v60,z5,tPen\WObj:=wPaper;
    MoveL Offs(pOrigin,292.71,103.70,6.00),vTravel,z5,tPen\WObj:=wPaper;
    MoveL Offs(pOrigin,292.71,103.70,0.00),v60,z0,tPen\WObj:=wPaper;
    MoveL Offs(pOrigin,293.77,103.70,0.00),v40,z0,tPen\WObj:=wPaper;
    MoveL Offs(pOrigin,294.62,102.87,0.00),v40,z0,tPen\WObj:=wPaper;
    MoveL Offs(pOrigin,292.07,105.43,0.00),v40,z0,tPen\WObj:=wPaper;
    MoveL Offs(pOrigin,292.92,104.76,0.00),v40,z0,tPen\WObj:=wPaper;
    MoveL Offs(pOrigin,294.41,104.76,0.00),v40,z0,tPen\WObj:=wPaper;
    MoveL Offs(pOrigin,295.07,103.92,0.00),v40,z0,tPen\WObj:=wPaper;
    MoveL Offs(pOrigin,292.37,106.62,0.00),v40,fine,tPen\WObj:=wPaper;
    MoveL Offs(pOrigin,292.37,106.62,6.00),v60,z5,tPen\WObj:=wPaper;
    MoveL Offs(pOrigin,292.66,107.82,6.00),vTravel,z5,tPen\WObj:=wPaper;
    MoveL Offs(pOrigin,292.66,107.82,0.00),v60,z0,tPen\WObj:=wPaper;
    MoveL Offs(pOrigin,296.12,104.37,0.00),v40,z0,tPen\WObj:=wPaper;
    MoveL Offs(pOrigin,296.14,105.27,0.00),v40,z0,tPen\WObj:=wPaper;
    MoveL Offs(pOrigin,297.64,106.78,0.00),v40,z0,tPen\WObj:=wPaper;
    MoveL Offs(pOrigin,297.17,106.15,0.00),v40,z0,tPen\WObj:=wPaper;
    MoveL Offs(pOrigin,296.11,105.94,0.00),v40,fine,tPen\WObj:=wPaper;
    MoveL Offs(pOrigin,296.11,105.94,6.00),v60,z5,tPen\WObj:=wPaper;
    MoveL Offs(pOrigin,299.10,107.35,6.00),vTravel,z5,tPen\WObj:=wPaper;
    MoveL Offs(pOrigin,299.10,107.35,0.00),v60,z0,tPen\WObj:=wPaper;
    MoveL Offs(pOrigin,301.06,105.40,0.00),v40,fine,tPen\WObj:=wPaper;
    MoveL Offs(pOrigin,301.06,105.40,6.00),v60,z5,tPen\WObj:=wPaper;
    MoveL Offs(pOrigin,302.70,108.24,6.00),vTravel,z5,tPen\WObj:=wPaper;
    MoveL Offs(pOrigin,302.70,108.24,0.00),v60,z0,tPen\WObj:=wPaper;
    MoveL Offs(pOrigin,304.65,106.29,0.00),v40,fine,tPen\WObj:=wPaper;
    MoveL Offs(pOrigin,304.65,106.29,6.00),v60,z5,tPen\WObj:=wPaper;
    MoveL Offs(pOrigin,306.29,109.13,6.00),vTravel,z5,tPen\WObj:=wPaper;
    MoveL Offs(pOrigin,306.29,109.13,0.00),v60,z0,tPen\WObj:=wPaper;
    MoveL Offs(pOrigin,308.24,107.17,0.00),v40,fine,tPen\WObj:=wPaper;
    MoveL Offs(pOrigin,308.24,107.17,6.00),v60,z5,tPen\WObj:=wPaper;
    MoveL Offs(pOrigin,310.03,109.87,6.00),vTravel,z5,tPen\WObj:=wPaper;
    MoveL Offs(pOrigin,310.03,109.87,0.00),v60,z0,tPen\WObj:=wPaper;
    MoveL Offs(pOrigin,311.99,107.91,0.00),v40,fine,tPen\WObj:=wPaper;
    MoveL Offs(pOrigin,311.99,107.91,6.00),v60,z5,tPen\WObj:=wPaper;
    MoveL Offs(pOrigin,314.23,108.65,6.00),vTravel,z5,tPen\WObj:=wPaper;
    MoveL Offs(pOrigin,314.23,108.65,0.00),v60,z0,tPen\WObj:=wPaper;
    MoveL Offs(pOrigin,312.28,110.61,0.00),v40,fine,tPen\WObj:=wPaper;
    MoveL Offs(pOrigin,312.28,110.61,6.00),v60,z5,tPen\WObj:=wPaper;
    MoveL Offs(pOrigin,314.67,111.20,6.00),vTravel,z5,tPen\WObj:=wPaper;
    MoveL Offs(pOrigin,314.67,111.20,0.00),v60,z0,tPen\WObj:=wPaper;
    MoveL Offs(pOrigin,316.63,109.25,0.00),v40,fine,tPen\WObj:=wPaper;
    MoveL Offs(pOrigin,316.63,109.25,6.00),v60,z5,tPen\WObj:=wPaper;
  ENDPROC

  PROC DrawPart202()
    MoveL Offs(pOrigin,318.26,112.09,6.00),vTravel,z5,tPen\WObj:=wPaper;
    MoveL Offs(pOrigin,318.26,112.09,0.00),v60,z0,tPen\WObj:=wPaper;
    MoveL Offs(pOrigin,320.22,110.13,0.00),v40,fine,tPen\WObj:=wPaper;
    MoveL Offs(pOrigin,320.22,110.13,6.00),v60,z5,tPen\WObj:=wPaper;
    MoveL Offs(pOrigin,326.50,114.31,6.00),vTravel,z5,tPen\WObj:=wPaper;
    MoveL Offs(pOrigin,326.50,114.31,0.00),v60,z0,tPen\WObj:=wPaper;
    MoveL Offs(pOrigin,328.45,112.36,0.00),v40,fine,tPen\WObj:=wPaper;
    MoveL Offs(pOrigin,328.45,112.36,6.00),v60,z5,tPen\WObj:=wPaper;
    MoveL Offs(pOrigin,330.84,112.95,6.00),vTravel,z5,tPen\WObj:=wPaper;
    MoveL Offs(pOrigin,330.84,112.95,0.00),v60,z0,tPen\WObj:=wPaper;
    MoveL Offs(pOrigin,328.89,114.90,0.00),v40,fine,tPen\WObj:=wPaper;
    MoveL Offs(pOrigin,328.89,114.90,6.00),v60,z5,tPen\WObj:=wPaper;
    MoveL Offs(pOrigin,331.14,115.64,6.00),vTravel,z5,tPen\WObj:=wPaper;
    MoveL Offs(pOrigin,331.14,115.64,0.00),v60,z0,tPen\WObj:=wPaper;
    MoveL Offs(pOrigin,333.09,113.69,0.00),v40,fine,tPen\WObj:=wPaper;
    MoveL Offs(pOrigin,333.09,113.69,6.00),v60,z5,tPen\WObj:=wPaper;
    MoveL Offs(pOrigin,334.73,116.53,6.00),vTravel,z5,tPen\WObj:=wPaper;
    MoveL Offs(pOrigin,334.73,116.53,0.00),v60,z0,tPen\WObj:=wPaper;
    MoveL Offs(pOrigin,336.68,114.58,0.00),v40,fine,tPen\WObj:=wPaper;
    MoveL Offs(pOrigin,336.68,114.58,6.00),v60,z5,tPen\WObj:=wPaper;
    MoveL Offs(pOrigin,338.78,115.47,6.00),vTravel,z5,tPen\WObj:=wPaper;
    MoveL Offs(pOrigin,338.78,115.47,0.00),v60,z0,tPen\WObj:=wPaper;
    MoveL Offs(pOrigin,336.82,117.42,0.00),v40,fine,tPen\WObj:=wPaper;
    MoveL Offs(pOrigin,336.82,117.42,6.00),v60,z5,tPen\WObj:=wPaper;
    MoveL Offs(pOrigin,339.22,118.01,6.00),vTravel,z5,tPen\WObj:=wPaper;
    MoveL Offs(pOrigin,339.22,118.01,0.00),v60,z0,tPen\WObj:=wPaper;
    MoveL Offs(pOrigin,341.17,116.06,0.00),v40,fine,tPen\WObj:=wPaper;
    MoveL Offs(pOrigin,341.17,116.06,6.00),v60,z5,tPen\WObj:=wPaper;
    MoveL Offs(pOrigin,343.42,116.80,6.00),vTravel,z5,tPen\WObj:=wPaper;
    MoveL Offs(pOrigin,343.42,116.80,0.00),v60,z0,tPen\WObj:=wPaper;
    MoveL Offs(pOrigin,341.61,118.61,0.00),v40,fine,tPen\WObj:=wPaper;
    MoveL Offs(pOrigin,341.61,118.61,6.00),v60,z5,tPen\WObj:=wPaper;
    MoveL Offs(pOrigin,343.41,119.80,6.00),vTravel,z5,tPen\WObj:=wPaper;
    MoveL Offs(pOrigin,343.41,119.80,0.00),v60,z0,tPen\WObj:=wPaper;
    MoveL Offs(pOrigin,345.51,117.70,0.00),v40,fine,tPen\WObj:=wPaper;
    MoveL Offs(pOrigin,345.51,117.70,6.00),v60,z5,tPen\WObj:=wPaper;
    MoveL Offs(pOrigin,349.54,122.63,6.00),vTravel,z5,tPen\WObj:=wPaper;
    MoveL Offs(pOrigin,349.54,122.63,0.00),v60,z0,tPen\WObj:=wPaper;
    MoveL Offs(pOrigin,353.00,119.17,0.00),v40,z0,tPen\WObj:=wPaper;
    MoveL Offs(pOrigin,353.44,120.22,0.00),v40,z0,tPen\WObj:=wPaper;
    MoveL Offs(pOrigin,349.69,123.97,0.00),v40,fine,tPen\WObj:=wPaper;
    MoveL Offs(pOrigin,349.69,123.97,6.00),v60,z5,tPen\WObj:=wPaper;
    MoveL Offs(pOrigin,349.98,125.17,6.00),vTravel,z5,tPen\WObj:=wPaper;
    MoveL Offs(pOrigin,349.98,125.17,0.00),v60,z0,tPen\WObj:=wPaper;
    MoveL Offs(pOrigin,353.89,121.27,0.00),v40,fine,tPen\WObj:=wPaper;
    MoveL Offs(pOrigin,353.89,121.27,6.00),v60,z5,tPen\WObj:=wPaper;
    MoveL Offs(pOrigin,354.93,123.21,6.00),vTravel,z5,tPen\WObj:=wPaper;
    MoveL Offs(pOrigin,354.93,123.21,0.00),v60,z0,tPen\WObj:=wPaper;
    MoveL Offs(pOrigin,350.42,127.72,0.00),v40,fine,tPen\WObj:=wPaper;
    MoveL Offs(pOrigin,350.42,127.72,6.00),v60,z5,tPen\WObj:=wPaper;
    MoveL Offs(pOrigin,351.79,129.05,6.00),vTravel,z5,tPen\WObj:=wPaper;
    MoveL Offs(pOrigin,351.79,129.05,0.00),v60,z0,tPen\WObj:=wPaper;
    MoveL Offs(pOrigin,354.34,129.05,0.00),v40,fine,tPen\WObj:=wPaper;
    MoveL Offs(pOrigin,354.34,129.05,6.00),v60,z5,tPen\WObj:=wPaper;
    MoveL Offs(pOrigin,354.12,132.22,6.00),vTravel,z5,tPen\WObj:=wPaper;
    MoveL Offs(pOrigin,354.12,132.22,0.00),v60,z0,tPen\WObj:=wPaper;
    MoveL Offs(pOrigin,352.42,132.22,0.00),v40,z0,tPen\WObj:=wPaper;
    MoveL Offs(pOrigin,352.64,133.27,0.00),v40,z0,tPen\WObj:=wPaper;
    MoveL Offs(pOrigin,354.12,133.27,0.00),v40,fine,tPen\WObj:=wPaper;
    MoveL Offs(pOrigin,354.12,133.27,6.00),v60,z5,tPen\WObj:=wPaper;
    MoveL Offs(pOrigin,354.55,135.38,6.00),vTravel,z5,tPen\WObj:=wPaper;
    MoveL Offs(pOrigin,354.55,135.38,0.00),v60,z0,tPen\WObj:=wPaper;
    MoveL Offs(pOrigin,353.06,135.38,0.00),v40,z0,tPen\WObj:=wPaper;
    MoveL Offs(pOrigin,352.05,135.05,0.00),v40,z0,tPen\WObj:=wPaper;
    MoveL Offs(pOrigin,358.21,128.89,0.00),v40,z0,tPen\WObj:=wPaper;
    MoveL Offs(pOrigin,357.76,127.84,0.00),v40,z0,tPen\WObj:=wPaper;
    MoveL Offs(pOrigin,351.75,133.85,0.00),v40,fine,tPen\WObj:=wPaper;
    MoveL Offs(pOrigin,351.75,133.85,6.00),v60,z5,tPen\WObj:=wPaper;
    MoveL Offs(pOrigin,351.16,131.46,6.00),vTravel,z5,tPen\WObj:=wPaper;
    MoveL Offs(pOrigin,351.16,131.46,0.00),v60,z0,tPen\WObj:=wPaper;
    MoveL Offs(pOrigin,356.57,126.05,0.00),v40,z0,tPen\WObj:=wPaper;
    MoveL Offs(pOrigin,355.97,125.15,0.00),v40,z0,tPen\WObj:=wPaper;
    MoveL Offs(pOrigin,351.01,130.11,0.00),v40,fine,tPen\WObj:=wPaper;
    MoveL Offs(pOrigin,351.01,130.11,6.00),v60,z5,tPen\WObj:=wPaper;
    MoveL Offs(pOrigin,345.79,128.04,6.00),vTravel,z5,tPen\WObj:=wPaper;
    MoveL Offs(pOrigin,345.79,128.04,0.00),v60,z0,tPen\WObj:=wPaper;
    MoveL Offs(pOrigin,344.29,126.54,0.00),v40,fine,tPen\WObj:=wPaper;
    MoveL Offs(pOrigin,344.29,126.54,6.00),v60,z5,tPen\WObj:=wPaper;
    MoveL Offs(pOrigin,341.60,129.83,6.00),vTravel,z5,tPen\WObj:=wPaper;
    MoveL Offs(pOrigin,341.60,129.83,0.00),v60,z0,tPen\WObj:=wPaper;
    MoveL Offs(pOrigin,339.05,127.28,0.00),v40,fine,tPen\WObj:=wPaper;
    MoveL Offs(pOrigin,339.05,127.28,6.00),v60,z5,tPen\WObj:=wPaper;
    MoveL Offs(pOrigin,337.70,128.92,6.00),vTravel,z5,tPen\WObj:=wPaper;
    MoveL Offs(pOrigin,337.70,128.92,0.00),v60,z0,tPen\WObj:=wPaper;
    MoveL Offs(pOrigin,335.00,126.21,0.00),v40,fine,tPen\WObj:=wPaper;
    MoveL Offs(pOrigin,335.00,126.21,6.00),v60,z5,tPen\WObj:=wPaper;
    MoveL Offs(pOrigin,334.84,124.57,6.00),vTravel,z5,tPen\WObj:=wPaper;
    MoveL Offs(pOrigin,334.84,124.57,0.00),v60,z0,tPen\WObj:=wPaper;
    MoveL Offs(pOrigin,333.94,123.66,0.00),v40,z0,tPen\WObj:=wPaper;
    MoveL Offs(pOrigin,334.41,122.82,0.00),v40,z0,tPen\WObj:=wPaper;
    MoveL Offs(pOrigin,330.20,127.03,0.00),v40,z0,tPen\WObj:=wPaper;
    MoveL Offs(pOrigin,331.11,126.80,0.00),v40,z0,tPen\WObj:=wPaper;
    MoveL Offs(pOrigin,328.55,124.25,0.00),v40,fine,tPen\WObj:=wPaper;
    MoveL Offs(pOrigin,328.55,124.25,6.00),v60,z5,tPen\WObj:=wPaper;
    MoveL Offs(pOrigin,326.91,125.59,6.00),vTravel,z5,tPen\WObj:=wPaper;
    MoveL Offs(pOrigin,326.91,125.59,0.00),v60,z0,tPen\WObj:=wPaper;
    MoveL Offs(pOrigin,324.20,122.89,0.00),v40,fine,tPen\WObj:=wPaper;
    MoveL Offs(pOrigin,324.20,122.89,6.00),v60,z5,tPen\WObj:=wPaper;
    MoveL Offs(pOrigin,324.66,124.83,6.00),vTravel,z5,tPen\WObj:=wPaper;
    MoveL Offs(pOrigin,324.66,124.83,0.00),v60,z0,tPen\WObj:=wPaper;
    MoveL Offs(pOrigin,322.25,122.43,0.00),v40,fine,tPen\WObj:=wPaper;
    MoveL Offs(pOrigin,322.25,122.43,6.00),v60,z5,tPen\WObj:=wPaper;
    MoveL Offs(pOrigin,325.56,125.70,6.00),vTravel,z5,tPen\WObj:=wPaper;
    MoveL Offs(pOrigin,325.56,125.70,0.00),v60,z0,tPen\WObj:=wPaper;
    MoveL Offs(pOrigin,329.62,121.64,0.00),v40,fine,tPen\WObj:=wPaper;
    MoveL Offs(pOrigin,329.62,121.64,6.00),v60,z5,tPen\WObj:=wPaper;
    MoveL Offs(pOrigin,330.82,121.94,6.00),vTravel,z5,tPen\WObj:=wPaper;
    MoveL Offs(pOrigin,330.82,121.94,0.00),v60,z0,tPen\WObj:=wPaper;
    MoveL Offs(pOrigin,326.76,125.99,0.00),v40,fine,tPen\WObj:=wPaper;
    MoveL Offs(pOrigin,326.76,125.99,6.00),v60,z5,tPen\WObj:=wPaper;
    MoveL Offs(pOrigin,329.00,126.73,6.00),vTravel,z5,tPen\WObj:=wPaper;
    MoveL Offs(pOrigin,329.00,126.73,0.00),v60,z0,tPen\WObj:=wPaper;
    MoveL Offs(pOrigin,333.06,122.68,0.00),v40,fine,tPen\WObj:=wPaper;
    MoveL Offs(pOrigin,333.06,122.68,6.00),v60,z5,tPen\WObj:=wPaper;
    MoveL Offs(pOrigin,335.46,123.27,6.00),vTravel,z5,tPen\WObj:=wPaper;
    MoveL Offs(pOrigin,335.46,123.27,0.00),v60,z0,tPen\WObj:=wPaper;
    MoveL Offs(pOrigin,331.40,127.33,0.00),v40,fine,tPen\WObj:=wPaper;
    MoveL Offs(pOrigin,331.40,127.33,6.00),v60,z5,tPen\WObj:=wPaper;
    MoveL Offs(pOrigin,333.34,128.37,6.00),vTravel,z5,tPen\WObj:=wPaper;
    MoveL Offs(pOrigin,333.34,128.37,0.00),v60,z0,tPen\WObj:=wPaper;
  ENDPROC

  PROC DrawPart203()
    MoveL Offs(pOrigin,337.85,123.86,0.00),v40,z0,tPen\WObj:=wPaper;
    MoveL Offs(pOrigin,338.90,124.31,0.00),v40,z0,tPen\WObj:=wPaper;
    MoveL Offs(pOrigin,334.09,129.12,0.00),v40,fine,tPen\WObj:=wPaper;
    MoveL Offs(pOrigin,334.09,129.12,6.00),v60,z5,tPen\WObj:=wPaper;
    MoveL Offs(pOrigin,336.70,130.16,6.00),vTravel,z5,tPen\WObj:=wPaper;
    MoveL Offs(pOrigin,336.70,130.16,0.00),v60,z0,tPen\WObj:=wPaper;
    MoveL Offs(pOrigin,337.12,130.59,0.00),v40,z0,tPen\WObj:=wPaper;
    MoveL Offs(pOrigin,336.70,130.16,0.00),v40,fine,tPen\WObj:=wPaper;
    MoveL Offs(pOrigin,336.70,130.16,6.00),v60,z5,tPen\WObj:=wPaper;
    MoveL Offs(pOrigin,352.49,137.60,6.00),vTravel,z5,tPen\WObj:=wPaper;
    MoveL Offs(pOrigin,352.49,137.60,0.00),v60,z0,tPen\WObj:=wPaper;
    MoveL Offs(pOrigin,359.70,130.39,0.00),v40,fine,tPen\WObj:=wPaper;
    MoveL Offs(pOrigin,359.70,130.39,6.00),v60,z5,tPen\WObj:=wPaper;
    MoveL Offs(pOrigin,359.01,136.54,6.00),vTravel,z5,tPen\WObj:=wPaper;
    MoveL Offs(pOrigin,359.01,136.54,0.00),v60,z0,tPen\WObj:=wPaper;
    MoveL Offs(pOrigin,359.65,136.54,0.00),v40,z0,tPen\WObj:=wPaper;
    MoveL Offs(pOrigin,360.50,137.39,0.00),v40,z0,tPen\WObj:=wPaper;
    MoveL Offs(pOrigin,360.50,138.24,0.00),v40,fine,tPen\WObj:=wPaper;
    MoveL Offs(pOrigin,360.50,138.24,6.00),v60,z5,tPen\WObj:=wPaper;
    MoveL Offs(pOrigin,359.01,137.39,6.00),vTravel,z5,tPen\WObj:=wPaper;
    MoveL Offs(pOrigin,359.01,137.39,0.00),v60,z0,tPen\WObj:=wPaper;
    MoveL Offs(pOrigin,359.44,137.81,0.00),v40,z0,tPen\WObj:=wPaper;
    MoveL Offs(pOrigin,359.01,137.39,0.00),v40,fine,tPen\WObj:=wPaper;
    MoveL Offs(pOrigin,359.01,137.39,6.00),v60,z5,tPen\WObj:=wPaper;
    MoveL Offs(pOrigin,356.67,140.88,6.00),vTravel,z5,tPen\WObj:=wPaper;
    MoveL Offs(pOrigin,356.67,140.88,0.00),v60,z0,tPen\WObj:=wPaper;
    MoveL Offs(pOrigin,354.12,143.43,0.00),v40,z0,tPen\WObj:=wPaper;
    MoveL Offs(pOrigin,354.98,142.78,0.00),v40,z0,tPen\WObj:=wPaper;
    MoveL Offs(pOrigin,356.04,142.78,0.00),v40,z0,tPen\WObj:=wPaper;
    MoveL Offs(pOrigin,355.83,141.72,0.00),v40,z0,tPen\WObj:=wPaper;
    MoveL Offs(pOrigin,354.55,141.72,0.00),v40,fine,tPen\WObj:=wPaper;
    MoveL Offs(pOrigin,354.55,141.72,6.00),v60,z5,tPen\WObj:=wPaper;
    MoveL Offs(pOrigin,356.97,142.08,6.00),vTravel,z5,tPen\WObj:=wPaper;
    MoveL Offs(pOrigin,356.97,142.08,0.00),v60,z0,tPen\WObj:=wPaper;
    MoveL Offs(pOrigin,354.27,144.78,0.00),v40,z0,tPen\WObj:=wPaper;
    MoveL Offs(pOrigin,354.71,145.83,0.00),v40,z0,tPen\WObj:=wPaper;
    MoveL Offs(pOrigin,357.27,143.28,0.00),v40,fine,tPen\WObj:=wPaper;
    MoveL Offs(pOrigin,357.27,143.28,6.00),v60,z5,tPen\WObj:=wPaper;
    MoveL Offs(pOrigin,357.56,144.47,6.00),vTravel,z5,tPen\WObj:=wPaper;
    MoveL Offs(pOrigin,357.56,144.47,0.00),v60,z0,tPen\WObj:=wPaper;
    MoveL Offs(pOrigin,354.86,147.18,0.00),v40,z0,tPen\WObj:=wPaper;
    MoveL Offs(pOrigin,355.83,147.00,0.00),v40,z0,tPen\WObj:=wPaper;
    MoveL Offs(pOrigin,357.10,147.00,0.00),v40,z0,tPen\WObj:=wPaper;
    MoveL Offs(pOrigin,357.31,148.06,0.00),v40,z0,tPen\WObj:=wPaper;
    MoveL Offs(pOrigin,356.25,148.06,0.00),v40,z0,tPen\WObj:=wPaper;
    MoveL Offs(pOrigin,355.59,148.30,0.00),v40,z0,tPen\WObj:=wPaper;
    MoveL Offs(pOrigin,358.59,151.30,0.00),v40,z0,tPen\WObj:=wPaper;
    MoveL Offs(pOrigin,358.16,151.22,0.00),v40,z0,tPen\WObj:=wPaper;
    MoveL Offs(pOrigin,357.10,151.22,0.00),v40,z0,tPen\WObj:=wPaper;
    MoveL Offs(pOrigin,357.31,152.28,0.00),v40,z0,tPen\WObj:=wPaper;
    MoveL Offs(pOrigin,358.38,152.28,0.00),v40,z0,tPen\WObj:=wPaper;
    MoveL Offs(pOrigin,359.19,151.81,0.00),v40,z0,tPen\WObj:=wPaper;
    MoveL Offs(pOrigin,356.63,154.36,0.00),v40,z0,tPen\WObj:=wPaper;
    MoveL Offs(pOrigin,357.26,154.44,0.00),v40,z0,tPen\WObj:=wPaper;
    MoveL Offs(pOrigin,360.11,157.30,0.00),v40,z0,tPen\WObj:=wPaper;
    MoveL Offs(pOrigin,359.65,157.56,0.00),v40,z0,tPen\WObj:=wPaper;
    MoveL Offs(pOrigin,358.59,157.56,0.00),v40,z0,tPen\WObj:=wPaper;
    MoveL Offs(pOrigin,357.67,157.80,0.00),v40,z0,tPen\WObj:=wPaper;
    MoveL Offs(pOrigin,360.07,155.40,0.00),v40,z0,tPen\WObj:=wPaper;
    MoveL Offs(pOrigin,359.65,155.35,0.00),v40,z0,tPen\WObj:=wPaper;
    MoveL Offs(pOrigin,356.65,152.35,0.00),v40,z0,tPen\WObj:=wPaper;
    MoveL Offs(pOrigin,356.19,151.82,0.00),v40,z0,tPen\WObj:=wPaper;
    MoveL Offs(pOrigin,358.60,149.41,0.00),v40,z0,tPen\WObj:=wPaper;
    MoveL Offs(pOrigin,357.95,150.17,0.00),v40,z0,tPen\WObj:=wPaper;
    MoveL Offs(pOrigin,356.67,150.17,0.00),v40,z0,tPen\WObj:=wPaper;
    MoveL Offs(pOrigin,356.19,150.40,0.00),v40,z0,tPen\WObj:=wPaper;
    MoveL Offs(pOrigin,359.20,153.40,0.00),v40,z0,tPen\WObj:=wPaper;
    MoveL Offs(pOrigin,359.48,153.01,0.00),v40,z0,tPen\WObj:=wPaper;
    MoveL Offs(pOrigin,357.08,155.41,0.00),v40,z0,tPen\WObj:=wPaper;
    MoveL Offs(pOrigin,358.16,155.45,0.00),v40,z0,tPen\WObj:=wPaper;
    MoveL Offs(pOrigin,359.22,155.45,0.00),v40,z0,tPen\WObj:=wPaper;
    MoveL Offs(pOrigin,359.44,156.50,0.00),v40,z0,tPen\WObj:=wPaper;
    MoveL Offs(pOrigin,358.38,156.50,0.00),v40,z0,tPen\WObj:=wPaper;
    MoveL Offs(pOrigin,357.71,156.39,0.00),v40,z0,tPen\WObj:=wPaper;
    MoveL Offs(pOrigin,360.72,159.40,0.00),v40,z0,tPen\WObj:=wPaper;
    MoveL Offs(pOrigin,360.29,159.67,0.00),v40,z0,tPen\WObj:=wPaper;
    MoveL Offs(pOrigin,359.22,159.67,0.00),v40,z0,tPen\WObj:=wPaper;
    MoveL Offs(pOrigin,358.77,160.44,0.00),v40,z0,tPen\WObj:=wPaper;
    MoveL Offs(pOrigin,361.78,163.45,0.00),v40,z0,tPen\WObj:=wPaper;
    MoveL Offs(pOrigin,362.30,163.63,0.00),v40,z0,tPen\WObj:=wPaper;
    MoveL Offs(pOrigin,359.89,166.04,0.00),v40,fine,tPen\WObj:=wPaper;
    MoveL Offs(pOrigin,359.89,166.04,6.00),v60,z5,tPen\WObj:=wPaper;
    MoveL Offs(pOrigin,360.74,166.89,6.00),vTravel,z5,tPen\WObj:=wPaper;
    MoveL Offs(pOrigin,360.74,166.89,0.00),v60,z0,tPen\WObj:=wPaper;
    MoveL Offs(pOrigin,363.44,169.59,0.00),v40,z0,tPen\WObj:=wPaper;
    MoveL Offs(pOrigin,363.93,169.47,0.00),v40,z0,tPen\WObj:=wPaper;
    MoveL Offs(pOrigin,361.67,171.72,0.00),v40,z0,tPen\WObj:=wPaper;
    MoveL Offs(pOrigin,361.65,170.79,0.00),v40,z0,tPen\WObj:=wPaper;
    MoveL Offs(pOrigin,364.65,173.79,0.00),v40,z0,tPen\WObj:=wPaper;
    MoveL Offs(pOrigin,365.26,174.11,0.00),v40,z0,tPen\WObj:=wPaper;
    MoveL Offs(pOrigin,363.01,176.36,0.00),v40,fine,tPen\WObj:=wPaper;
    MoveL Offs(pOrigin,363.01,176.36,6.00),v60,z5,tPen\WObj:=wPaper;
    MoveL Offs(pOrigin,362.71,175.17,6.00),vTravel,z5,tPen\WObj:=wPaper;
    MoveL Offs(pOrigin,362.71,175.17,0.00),v60,z0,tPen\WObj:=wPaper;
    MoveL Offs(pOrigin,364.81,173.06,0.00),v40,fine,tPen\WObj:=wPaper;
    MoveL Offs(pOrigin,364.81,173.06,6.00),v60,z5,tPen\WObj:=wPaper;
    MoveL Offs(pOrigin,364.67,171.71,6.00),vTravel,z5,tPen\WObj:=wPaper;
    MoveL Offs(pOrigin,364.67,171.71,0.00),v60,z0,tPen\WObj:=wPaper;
    MoveL Offs(pOrigin,362.26,174.12,0.00),v40,z0,tPen\WObj:=wPaper;
    MoveL Offs(pOrigin,362.86,174.98,0.00),v40,z0,tPen\WObj:=wPaper;
    MoveL Offs(pOrigin,365.87,177.99,0.00),v40,z0,tPen\WObj:=wPaper;
    MoveL Offs(pOrigin,366.45,177.40,0.00),v40,z0,tPen\WObj:=wPaper;
    MoveL Offs(pOrigin,364.19,179.66,0.00),v40,z0,tPen\WObj:=wPaper;
    MoveL Offs(pOrigin,364.52,179.63,0.00),v40,z0,tPen\WObj:=wPaper;
    MoveL Offs(pOrigin,367.68,182.79,0.00),v40,z0,tPen\WObj:=wPaper;
    MoveL Offs(pOrigin,368.38,182.94,0.00),v40,z0,tPen\WObj:=wPaper;
    MoveL Offs(pOrigin,366.28,185.04,0.00),v40,z0,tPen\WObj:=wPaper;
    MoveL Offs(pOrigin,366.49,184.58,0.00),v40,z0,tPen\WObj:=wPaper;
    MoveL Offs(pOrigin,374.30,192.40,0.00),v40,z0,tPen\WObj:=wPaper;
    MoveL Offs(pOrigin,374.94,192.80,0.00),v40,z0,tPen\WObj:=wPaper;
    MoveL Offs(pOrigin,372.69,195.06,0.00),v40,z0,tPen\WObj:=wPaper;
    MoveL Offs(pOrigin,372.96,194.04,0.00),v40,z0,tPen\WObj:=wPaper;
    MoveL Offs(pOrigin,375.36,196.44,0.00),v40,z0,tPen\WObj:=wPaper;
    MoveL Offs(pOrigin,375.83,196.40,0.00),v40,z0,tPen\WObj:=wPaper;
    MoveL Offs(pOrigin,373.27,198.95,0.00),v40,z0,tPen\WObj:=wPaper;
    MoveL Offs(pOrigin,374.02,199.59,0.00),v40,z0,tPen\WObj:=wPaper;
    MoveL Offs(pOrigin,376.43,201.99,0.00),v40,z0,tPen\WObj:=wPaper;
    MoveL Offs(pOrigin,376.71,201.49,0.00),v40,z0,tPen\WObj:=wPaper;
    MoveL Offs(pOrigin,374.31,203.89,0.00),v40,z0,tPen\WObj:=wPaper;
    MoveL Offs(pOrigin,374.63,203.18,0.00),v40,z0,tPen\WObj:=wPaper;
  ENDPROC

  PROC DrawPart204()
    MoveL Offs(pOrigin,377.04,205.59,0.00),v40,z0,tPen\WObj:=wPaper;
    MoveL Offs(pOrigin,377.45,205.23,0.00),v40,z0,tPen\WObj:=wPaper;
    MoveL Offs(pOrigin,374.74,207.93,0.00),v40,fine,tPen\WObj:=wPaper;
    MoveL Offs(pOrigin,374.74,207.93,6.00),v60,z5,tPen\WObj:=wPaper;
    MoveL Offs(pOrigin,374.74,209.43,6.00),vTravel,z5,tPen\WObj:=wPaper;
    MoveL Offs(pOrigin,374.74,209.43,0.00),v60,z0,tPen\WObj:=wPaper;
    MoveL Offs(pOrigin,377.59,206.58,0.00),v40,z0,tPen\WObj:=wPaper;
    MoveL Offs(pOrigin,377.19,207.24,0.00),v40,z0,tPen\WObj:=wPaper;
    MoveL Offs(pOrigin,375.09,205.13,0.00),v40,z0,tPen\WObj:=wPaper;
    MoveL Offs(pOrigin,374.45,205.24,0.00),v40,z0,tPen\WObj:=wPaper;
    MoveL Offs(pOrigin,377.01,202.68,0.00),v40,fine,tPen\WObj:=wPaper;
    MoveL Offs(pOrigin,377.01,202.68,6.00),v60,z5,tPen\WObj:=wPaper;
    MoveL Offs(pOrigin,379.11,202.08,6.00),vTravel,z5,tPen\WObj:=wPaper;
    MoveL Offs(pOrigin,379.11,202.08,0.00),v60,z0,tPen\WObj:=wPaper;
    MoveL Offs(pOrigin,381.66,199.52,0.00),v40,z0,tPen\WObj:=wPaper;
    MoveL Offs(pOrigin,381.06,199.16,0.00),v40,z0,tPen\WObj:=wPaper;
    MoveL Offs(pOrigin,379.26,197.35,0.00),v40,z0,tPen\WObj:=wPaper;
    MoveL Offs(pOrigin,378.67,198.04,0.00),v40,z0,tPen\WObj:=wPaper;
    MoveL Offs(pOrigin,381.07,195.63,0.00),v40,z0,tPen\WObj:=wPaper;
    MoveL Offs(pOrigin,380.45,195.56,0.00),v40,z0,tPen\WObj:=wPaper;
    MoveL Offs(pOrigin,378.80,193.91,0.00),v40,z0,tPen\WObj:=wPaper;
    MoveL Offs(pOrigin,378.23,193.99,0.00),v40,z0,tPen\WObj:=wPaper;
    MoveL Offs(pOrigin,380.64,191.59,0.00),v40,z0,tPen\WObj:=wPaper;
    MoveL Offs(pOrigin,379.99,192.11,0.00),v40,z0,tPen\WObj:=wPaper;
    MoveL Offs(pOrigin,378.34,190.46,0.00),v40,z0,tPen\WObj:=wPaper;
    MoveL Offs(pOrigin,378.09,191.15,0.00),v40,z0,tPen\WObj:=wPaper;
    MoveL Offs(pOrigin,380.04,189.19,0.00),v40,z0,tPen\WObj:=wPaper;
    MoveL Offs(pOrigin,379.54,190.17,0.00),v40,z0,tPen\WObj:=wPaper;
    MoveL Offs(pOrigin,378.18,188.81,0.00),v40,z0,tPen\WObj:=wPaper;
    MoveL Offs(pOrigin,377.50,188.75,0.00),v40,z0,tPen\WObj:=wPaper;
    MoveL Offs(pOrigin,379.60,186.65,0.00),v40,z0,tPen\WObj:=wPaper;
    MoveL Offs(pOrigin,378.93,186.57,0.00),v40,z0,tPen\WObj:=wPaper;
    MoveL Offs(pOrigin,376.07,183.71,0.00),v40,z0,tPen\WObj:=wPaper;
    MoveL Offs(pOrigin,376.65,183.96,0.00),v40,z0,tPen\WObj:=wPaper;
    MoveL Offs(pOrigin,378.35,183.96,0.00),v40,z0,tPen\WObj:=wPaper;
    MoveL Offs(pOrigin,378.77,183.42,0.00),v40,z0,tPen\WObj:=wPaper;
    MoveL Offs(pOrigin,376.96,181.62,0.00),v40,fine,tPen\WObj:=wPaper;
    MoveL Offs(pOrigin,376.96,181.62,6.00),v60,z5,tPen\WObj:=wPaper;
    MoveL Offs(pOrigin,376.67,182.82,6.00),vTravel,z5,tPen\WObj:=wPaper;
    MoveL Offs(pOrigin,376.67,182.82,0.00),v60,z0,tPen\WObj:=wPaper;
    MoveL Offs(pOrigin,379.07,185.22,0.00),v40,z0,tPen\WObj:=wPaper;
    MoveL Offs(pOrigin,379.46,185.30,0.00),v40,z0,tPen\WObj:=wPaper;
    MoveL Offs(pOrigin,372.09,192.66,0.00),v40,z0,tPen\WObj:=wPaper;
    MoveL Offs(pOrigin,371.50,191.77,0.00),v40,z0,tPen\WObj:=wPaper;
    MoveL Offs(pOrigin,379.31,183.95,0.00),v40,fine,tPen\WObj:=wPaper;
    MoveL Offs(pOrigin,379.31,183.95,6.00),v60,z5,tPen\WObj:=wPaper;
    MoveL Offs(pOrigin,378.35,182.90,6.00),vTravel,z5,tPen\WObj:=wPaper;
    MoveL Offs(pOrigin,378.35,182.90,0.00),v60,z0,tPen\WObj:=wPaper;
    MoveL Offs(pOrigin,377.08,182.90,0.00),v40,fine,tPen\WObj:=wPaper;
    MoveL Offs(pOrigin,377.08,182.90,6.00),v60,z5,tPen\WObj:=wPaper;
    MoveL Offs(pOrigin,377.01,184.35,6.00),vTravel,z5,tPen\WObj:=wPaper;
    MoveL Offs(pOrigin,377.01,184.35,0.00),v60,z0,tPen\WObj:=wPaper;
    MoveL Offs(pOrigin,377.01,186.05,0.00),v40,fine,tPen\WObj:=wPaper;
    MoveL Offs(pOrigin,377.01,186.05,6.00),v60,z5,tPen\WObj:=wPaper;
    MoveL Offs(pOrigin,375.38,184.99,6.00),vTravel,z5,tPen\WObj:=wPaper;
    MoveL Offs(pOrigin,375.38,184.99,0.00),v60,z0,tPen\WObj:=wPaper;
    MoveL Offs(pOrigin,376.23,184.92,0.00),v40,z0,tPen\WObj:=wPaper;
    MoveL Offs(pOrigin,376.65,184.14,0.00),v40,z0,tPen\WObj:=wPaper;
    MoveL Offs(pOrigin,378.14,176.70,0.00),v40,z0,tPen\WObj:=wPaper;
    MoveL Offs(pOrigin,380.05,171.60,0.00),v40,z0,tPen\WObj:=wPaper;
    MoveL Offs(pOrigin,380.05,169.48,0.00),v40,z0,tPen\WObj:=wPaper;
    MoveL Offs(pOrigin,378.85,166.50,0.00),v40,z0,tPen\WObj:=wPaper;
    MoveL Offs(pOrigin,377.29,164.16,0.00),v40,z0,tPen\WObj:=wPaper;
    MoveL Offs(pOrigin,365.39,148.86,0.00),v40,z0,tPen\WObj:=wPaper;
    MoveL Offs(pOrigin,365.39,148.86,0.00),v40,z0,tPen\WObj:=wPaper;
    MoveL Offs(pOrigin,364.75,148.23,0.00),v40,z0,tPen\WObj:=wPaper;
    MoveL Offs(pOrigin,364.54,147.38,0.00),v40,fine,tPen\WObj:=wPaper;
    MoveL Offs(pOrigin,364.54,147.38,6.00),v60,z5,tPen\WObj:=wPaper;
    MoveL Offs(pOrigin,363.24,147.75,6.00),vTravel,z5,tPen\WObj:=wPaper;
    MoveL Offs(pOrigin,363.24,147.75,0.00),v60,z0,tPen\WObj:=wPaper;
    MoveL Offs(pOrigin,367.45,143.54,0.00),v40,z0,tPen\WObj:=wPaper;
    MoveL Offs(pOrigin,368.35,144.14,0.00),v40,z0,tPen\WObj:=wPaper;
    MoveL Offs(pOrigin,363.84,148.65,0.00),v40,z0,tPen\WObj:=wPaper;
    MoveL Offs(pOrigin,364.59,149.39,0.00),v40,z0,tPen\WObj:=wPaper;
    MoveL Offs(pOrigin,366.54,147.44,0.00),v40,z0,tPen\WObj:=wPaper;
    MoveL Offs(pOrigin,367.14,148.34,0.00),v40,z0,tPen\WObj:=wPaper;
    MoveL Offs(pOrigin,365.33,150.14,0.00),v40,z0,tPen\WObj:=wPaper;
    MoveL Offs(pOrigin,365.60,149.50,0.00),v40,z0,tPen\WObj:=wPaper;
    MoveL Offs(pOrigin,366.02,149.93,0.00),v40,z0,tPen\WObj:=wPaper;
    MoveL Offs(pOrigin,365.60,149.50,0.00),v40,fine,tPen\WObj:=wPaper;
    MoveL Offs(pOrigin,365.60,149.50,6.00),v60,z5,tPen\WObj:=wPaper;
    MoveL Offs(pOrigin,365.93,151.04,6.00),vTravel,z5,tPen\WObj:=wPaper;
    MoveL Offs(pOrigin,365.93,151.04,0.00),v60,z0,tPen\WObj:=wPaper;
    MoveL Offs(pOrigin,367.88,149.08,0.00),v40,z0,tPen\WObj:=wPaper;
    MoveL Offs(pOrigin,367.30,149.50,0.00),v40,z0,tPen\WObj:=wPaper;
    MoveL Offs(pOrigin,367.51,149.93,0.00),v40,z0,tPen\WObj:=wPaper;
    MoveL Offs(pOrigin,367.30,149.50,0.00),v40,fine,tPen\WObj:=wPaper;
    MoveL Offs(pOrigin,367.30,149.50,6.00),v60,z5,tPen\WObj:=wPaper;
    MoveL Offs(pOrigin,368.48,149.98,6.00),vTravel,z5,tPen\WObj:=wPaper;
    MoveL Offs(pOrigin,368.48,149.98,0.00),v60,z0,tPen\WObj:=wPaper;
    MoveL Offs(pOrigin,366.53,151.94,0.00),v40,z0,tPen\WObj:=wPaper;
    MoveL Offs(pOrigin,367.09,151.41,0.00),v40,z0,tPen\WObj:=wPaper;
    MoveL Offs(pOrigin,367.51,151.84,0.00),v40,z0,tPen\WObj:=wPaper;
    MoveL Offs(pOrigin,367.09,151.41,0.00),v40,fine,tPen\WObj:=wPaper;
    MoveL Offs(pOrigin,367.09,151.41,6.00),v60,z5,tPen\WObj:=wPaper;
    MoveL Offs(pOrigin,368.15,150.56,6.00),vTravel,z5,tPen\WObj:=wPaper;
    MoveL Offs(pOrigin,368.15,150.56,0.00),v60,z0,tPen\WObj:=wPaper;
    MoveL Offs(pOrigin,368.58,150.99,0.00),v40,z0,tPen\WObj:=wPaper;
    MoveL Offs(pOrigin,368.15,150.56,0.00),v40,z0,tPen\WObj:=wPaper;
    MoveL Offs(pOrigin,368.79,151.41,0.00),v40,z0,tPen\WObj:=wPaper;
    MoveL Offs(pOrigin,369.64,152.26,0.00),v40,z0,tPen\WObj:=wPaper;
    MoveL Offs(pOrigin,368.79,151.41,0.00),v40,z0,tPen\WObj:=wPaper;
    MoveL Offs(pOrigin,369.23,150.73,0.00),v40,z0,tPen\WObj:=wPaper;
    MoveL Offs(pOrigin,367.12,152.83,0.00),v40,z0,tPen\WObj:=wPaper;
    MoveL Offs(pOrigin,367.94,152.48,0.00),v40,z0,tPen\WObj:=wPaper;
    MoveL Offs(pOrigin,368.36,152.90,0.00),v40,z0,tPen\WObj:=wPaper;
    MoveL Offs(pOrigin,367.94,152.48,0.00),v40,fine,tPen\WObj:=wPaper;
    MoveL Offs(pOrigin,367.94,152.48,6.00),v60,z5,tPen\WObj:=wPaper;
    MoveL Offs(pOrigin,368.79,153.54,6.00),vTravel,z5,tPen\WObj:=wPaper;
    MoveL Offs(pOrigin,368.79,153.54,0.00),v60,z0,tPen\WObj:=wPaper;
    MoveL Offs(pOrigin,369.21,153.96,0.00),v40,z0,tPen\WObj:=wPaper;
    MoveL Offs(pOrigin,368.79,153.54,0.00),v40,z0,tPen\WObj:=wPaper;
    MoveL Offs(pOrigin,369.21,153.34,0.00),v40,z0,tPen\WObj:=wPaper;
    MoveL Offs(pOrigin,370.28,153.34,0.00),v40,z0,tPen\WObj:=wPaper;
    MoveL Offs(pOrigin,370.57,152.37,0.00),v40,z0,tPen\WObj:=wPaper;
    MoveL Offs(pOrigin,368.47,154.48,0.00),v40,z0,tPen\WObj:=wPaper;
    MoveL Offs(pOrigin,369.21,155.22,0.00),v40,z0,tPen\WObj:=wPaper;
    MoveL Offs(pOrigin,371.32,153.12,0.00),v40,z0,tPen\WObj:=wPaper;
    MoveL Offs(pOrigin,371.91,154.02,0.00),v40,z0,tPen\WObj:=wPaper;
    MoveL Offs(pOrigin,369.96,155.97,0.00),v40,z0,tPen\WObj:=wPaper;
  ENDPROC

  PROC DrawPart205()
    MoveL Offs(pOrigin,370.06,155.24,0.00),v40,z0,tPen\WObj:=wPaper;
    MoveL Offs(pOrigin,370.70,155.88,0.00),v40,z0,tPen\WObj:=wPaper;
    MoveL Offs(pOrigin,370.06,155.24,0.00),v40,z0,tPen\WObj:=wPaper;
    MoveL Offs(pOrigin,370.70,155.45,0.00),v40,z0,tPen\WObj:=wPaper;
    MoveL Offs(pOrigin,371.76,155.45,0.00),v40,z0,tPen\WObj:=wPaper;
    MoveL Offs(pOrigin,371.98,155.24,0.00),v40,z0,tPen\WObj:=wPaper;
    MoveL Offs(pOrigin,372.83,156.09,0.00),v40,z0,tPen\WObj:=wPaper;
    MoveL Offs(pOrigin,371.98,155.24,0.00),v40,z0,tPen\WObj:=wPaper;
    MoveL Offs(pOrigin,372.51,154.91,0.00),v40,z0,tPen\WObj:=wPaper;
    MoveL Offs(pOrigin,370.56,156.87,0.00),v40,z0,tPen\WObj:=wPaper;
    MoveL Offs(pOrigin,371.12,156.51,0.00),v40,z0,tPen\WObj:=wPaper;
    MoveL Offs(pOrigin,371.55,156.94,0.00),v40,z0,tPen\WObj:=wPaper;
    MoveL Offs(pOrigin,371.12,156.51,0.00),v40,z0,tPen\WObj:=wPaper;
    MoveL Offs(pOrigin,371.55,156.50,0.00),v40,z0,tPen\WObj:=wPaper;
    MoveL Offs(pOrigin,372.61,156.50,0.00),v40,z0,tPen\WObj:=wPaper;
    MoveL Offs(pOrigin,373.04,156.30,0.00),v40,z0,tPen\WObj:=wPaper;
    MoveL Offs(pOrigin,373.89,157.36,0.00),v40,z0,tPen\WObj:=wPaper;
    MoveL Offs(pOrigin,373.04,156.30,0.00),v40,z0,tPen\WObj:=wPaper;
    MoveL Offs(pOrigin,373.41,155.51,0.00),v40,z0,tPen\WObj:=wPaper;
    MoveL Offs(pOrigin,371.15,157.76,0.00),v40,z0,tPen\WObj:=wPaper;
    MoveL Offs(pOrigin,371.90,158.51,0.00),v40,z0,tPen\WObj:=wPaper;
    MoveL Offs(pOrigin,374.00,156.41,0.00),v40,z0,tPen\WObj:=wPaper;
    MoveL Offs(pOrigin,374.60,157.30,0.00),v40,z0,tPen\WObj:=wPaper;
    MoveL Offs(pOrigin,372.50,159.41,0.00),v40,z0,tPen\WObj:=wPaper;
    MoveL Offs(pOrigin,373.25,159.06,0.00),v40,z0,tPen\WObj:=wPaper;
    MoveL Offs(pOrigin,373.46,159.49,0.00),v40,z0,tPen\WObj:=wPaper;
    MoveL Offs(pOrigin,373.25,159.06,0.00),v40,z0,tPen\WObj:=wPaper;
    MoveL Offs(pOrigin,373.25,158.62,0.00),v40,z0,tPen\WObj:=wPaper;
    MoveL Offs(pOrigin,374.31,158.62,0.00),v40,z0,tPen\WObj:=wPaper;
    MoveL Offs(pOrigin,374.31,158.00,0.00),v40,z0,tPen\WObj:=wPaper;
    MoveL Offs(pOrigin,374.74,158.43,0.00),v40,z0,tPen\WObj:=wPaper;
    MoveL Offs(pOrigin,374.31,158.00,0.00),v40,z0,tPen\WObj:=wPaper;
    MoveL Offs(pOrigin,373.46,157.56,0.00),v40,z0,tPen\WObj:=wPaper;
    MoveL Offs(pOrigin,372.40,157.56,0.00),v40,z0,tPen\WObj:=wPaper;
    MoveL Offs(pOrigin,372.40,158.00,0.00),v40,z0,tPen\WObj:=wPaper;
    MoveL Offs(pOrigin,372.61,158.43,0.00),v40,z0,tPen\WObj:=wPaper;
    MoveL Offs(pOrigin,372.40,158.00,0.00),v40,fine,tPen\WObj:=wPaper;
    MoveL Offs(pOrigin,372.40,158.00,6.00),v60,z5,tPen\WObj:=wPaper;
    MoveL Offs(pOrigin,373.09,160.30,6.00),vTravel,z5,tPen\WObj:=wPaper;
    MoveL Offs(pOrigin,373.09,160.30,0.00),v60,z0,tPen\WObj:=wPaper;
    MoveL Offs(pOrigin,375.35,158.05,0.00),v40,z0,tPen\WObj:=wPaper;
    MoveL Offs(pOrigin,375.16,159.06,0.00),v40,z0,tPen\WObj:=wPaper;
    MoveL Offs(pOrigin,375.80,159.70,0.00),v40,z0,tPen\WObj:=wPaper;
    MoveL Offs(pOrigin,375.16,159.06,0.00),v40,z0,tPen\WObj:=wPaper;
    MoveL Offs(pOrigin,375.94,158.95,0.00),v40,z0,tPen\WObj:=wPaper;
    MoveL Offs(pOrigin,373.84,161.05,0.00),v40,z0,tPen\WObj:=wPaper;
    MoveL Offs(pOrigin,374.44,161.95,0.00),v40,z0,tPen\WObj:=wPaper;
    MoveL Offs(pOrigin,376.69,159.69,0.00),v40,z0,tPen\WObj:=wPaper;
    MoveL Offs(pOrigin,377.29,160.59,0.00),v40,z0,tPen\WObj:=wPaper;
    MoveL Offs(pOrigin,375.03,162.84,0.00),v40,z0,tPen\WObj:=wPaper;
    MoveL Offs(pOrigin,375.78,163.59,0.00),v40,z0,tPen\WObj:=wPaper;
    MoveL Offs(pOrigin,377.88,161.49,0.00),v40,z0,tPen\WObj:=wPaper;
    MoveL Offs(pOrigin,377.50,162.04,0.00),v40,z0,tPen\WObj:=wPaper;
    MoveL Offs(pOrigin,377.92,162.46,0.00),v40,z0,tPen\WObj:=wPaper;
    MoveL Offs(pOrigin,377.50,162.04,0.00),v40,z0,tPen\WObj:=wPaper;
    MoveL Offs(pOrigin,376.86,161.78,0.00),v40,z0,tPen\WObj:=wPaper;
    MoveL Offs(pOrigin,375.80,161.78,0.00),v40,fine,tPen\WObj:=wPaper;
    MoveL Offs(pOrigin,375.80,161.78,6.00),v60,z5,tPen\WObj:=wPaper;
    MoveL Offs(pOrigin,376.65,162.84,6.00),vTravel,z5,tPen\WObj:=wPaper;
    MoveL Offs(pOrigin,376.65,162.84,0.00),v60,z0,tPen\WObj:=wPaper;
    MoveL Offs(pOrigin,377.71,162.84,0.00),v40,z0,tPen\WObj:=wPaper;
    MoveL Offs(pOrigin,377.29,163.90,0.00),v40,z0,tPen\WObj:=wPaper;
    MoveL Offs(pOrigin,380.90,163.90,0.00),v40,z0,tPen\WObj:=wPaper;
    MoveL Offs(pOrigin,381.55,163.81,0.00),v40,z0,tPen\WObj:=wPaper;
    MoveL Offs(pOrigin,379.75,162.00,0.00),v40,z0,tPen\WObj:=wPaper;
    MoveL Offs(pOrigin,380.26,161.78,0.00),v40,z0,tPen\WObj:=wPaper;
    MoveL Offs(pOrigin,381.54,161.78,0.00),v40,fine,tPen\WObj:=wPaper;
    MoveL Offs(pOrigin,381.54,161.78,6.00),v60,z5,tPen\WObj:=wPaper;
    MoveL Offs(pOrigin,382.37,162.97,6.00),vTravel,z5,tPen\WObj:=wPaper;
    MoveL Offs(pOrigin,382.37,162.97,0.00),v60,z0,tPen\WObj:=wPaper;
    MoveL Offs(pOrigin,378.16,167.18,0.00),v40,z0,tPen\WObj:=wPaper;
    MoveL Offs(pOrigin,377.72,166.13,0.00),v40,z0,tPen\WObj:=wPaper;
    MoveL Offs(pOrigin,383.28,160.57,0.00),v40,z0,tPen\WObj:=wPaper;
    MoveL Offs(pOrigin,383.19,159.47,0.00),v40,z0,tPen\WObj:=wPaper;
    MoveL Offs(pOrigin,381.38,157.66,0.00),v40,z0,tPen\WObj:=wPaper;
    MoveL Offs(pOrigin,381.75,157.57,0.00),v40,z0,tPen\WObj:=wPaper;
    MoveL Offs(pOrigin,381.54,158.00,0.00),v40,z0,tPen\WObj:=wPaper;
    MoveL Offs(pOrigin,381.75,157.57,0.00),v40,z0,tPen\WObj:=wPaper;
    MoveL Offs(pOrigin,382.17,157.56,0.00),v40,z0,tPen\WObj:=wPaper;
    MoveL Offs(pOrigin,383.45,157.56,0.00),v40,z0,tPen\WObj:=wPaper;
    MoveL Offs(pOrigin,383.45,157.79,0.00),v40,z0,tPen\WObj:=wPaper;
    MoveL Offs(pOrigin,383.24,158.21,0.00),v40,z0,tPen\WObj:=wPaper;
    MoveL Offs(pOrigin,383.45,157.79,0.00),v40,z0,tPen\WObj:=wPaper;
    MoveL Offs(pOrigin,384.08,157.37,0.00),v40,z0,tPen\WObj:=wPaper;
    MoveL Offs(pOrigin,382.43,155.72,0.00),v40,z0,tPen\WObj:=wPaper;
    MoveL Offs(pOrigin,382.81,155.45,0.00),v40,z0,tPen\WObj:=wPaper;
    MoveL Offs(pOrigin,382.60,155.88,0.00),v40,z0,tPen\WObj:=wPaper;
    MoveL Offs(pOrigin,382.81,155.45,0.00),v40,z0,tPen\WObj:=wPaper;
    MoveL Offs(pOrigin,383.24,155.45,0.00),v40,z0,tPen\WObj:=wPaper;
    MoveL Offs(pOrigin,384.51,155.45,0.00),v40,z0,tPen\WObj:=wPaper;
    MoveL Offs(pOrigin,384.51,155.66,0.00),v40,z0,tPen\WObj:=wPaper;
    MoveL Offs(pOrigin,384.30,156.09,0.00),v40,z0,tPen\WObj:=wPaper;
    MoveL Offs(pOrigin,384.51,155.66,0.00),v40,z0,tPen\WObj:=wPaper;
    MoveL Offs(pOrigin,385.12,155.43,0.00),v40,z0,tPen\WObj:=wPaper;
    MoveL Offs(pOrigin,383.32,153.63,0.00),v40,z0,tPen\WObj:=wPaper;
    MoveL Offs(pOrigin,382.40,153.98,0.00),v40,z0,tPen\WObj:=wPaper;
    MoveL Offs(pOrigin,387.81,148.57,0.00),v40,z0,tPen\WObj:=wPaper;
    MoveL Offs(pOrigin,387.35,148.69,0.00),v40,z0,tPen\WObj:=wPaper;
    MoveL Offs(pOrigin,375.78,137.12,0.00),v40,z0,tPen\WObj:=wPaper;
    MoveL Offs(pOrigin,375.59,136.75,0.00),v40,z0,tPen\WObj:=wPaper;
    MoveL Offs(pOrigin,376.01,137.18,0.00),v40,z0,tPen\WObj:=wPaper;
    MoveL Offs(pOrigin,375.59,136.75,0.00),v40,z0,tPen\WObj:=wPaper;
    MoveL Offs(pOrigin,374.96,137.53,0.00),v40,z0,tPen\WObj:=wPaper;
    MoveL Offs(pOrigin,378.12,134.37,0.00),v40,z0,tPen\WObj:=wPaper;
    MoveL Offs(pOrigin,379.16,134.82,0.00),v40,z0,tPen\WObj:=wPaper;
    MoveL Offs(pOrigin,375.71,138.28,0.00),v40,z0,tPen\WObj:=wPaper;
    MoveL Offs(pOrigin,376.45,139.02,0.00),v40,z0,tPen\WObj:=wPaper;
    MoveL Offs(pOrigin,380.36,135.12,0.00),v40,z0,tPen\WObj:=wPaper;
    MoveL Offs(pOrigin,381.41,135.56,0.00),v40,z0,tPen\WObj:=wPaper;
    MoveL Offs(pOrigin,379.90,137.06,0.00),v40,z0,tPen\WObj:=wPaper;
    MoveL Offs(pOrigin,380.95,137.51,0.00),v40,z0,tPen\WObj:=wPaper;
    MoveL Offs(pOrigin,382.60,135.86,0.00),v40,z0,tPen\WObj:=wPaper;
    MoveL Offs(pOrigin,382.82,136.70,0.00),v40,z0,tPen\WObj:=wPaper;
    MoveL Offs(pOrigin,383.57,137.45,0.00),v40,z0,tPen\WObj:=wPaper;
    MoveL Offs(pOrigin,383.20,138.25,0.00),v40,z0,tPen\WObj:=wPaper;
    MoveL Offs(pOrigin,385.00,136.45,0.00),v40,fine,tPen\WObj:=wPaper;
    MoveL Offs(pOrigin,385.00,136.45,6.00),v60,z5,tPen\WObj:=wPaper;
    MoveL Offs(pOrigin,383.80,136.15,6.00),vTravel,z5,tPen\WObj:=wPaper;
    MoveL Offs(pOrigin,383.80,136.15,0.00),v60,z0,tPen\WObj:=wPaper;
    MoveL Offs(pOrigin,382.15,137.81,0.00),v40,fine,tPen\WObj:=wPaper;
  ENDPROC

  PROC DrawPart206()
    MoveL Offs(pOrigin,382.15,137.81,6.00),v60,z5,tPen\WObj:=wPaper;
    MoveL Offs(pOrigin,380.65,139.31,6.00),vTravel,z5,tPen\WObj:=wPaper;
    MoveL Offs(pOrigin,380.65,139.31,0.00),v60,z0,tPen\WObj:=wPaper;
    MoveL Offs(pOrigin,378.84,141.11,0.00),v40,z0,tPen\WObj:=wPaper;
    MoveL Offs(pOrigin,379.62,141.00,0.00),v40,z0,tPen\WObj:=wPaper;
    MoveL Offs(pOrigin,380.05,141.21,0.00),v40,z0,tPen\WObj:=wPaper;
    MoveL Offs(pOrigin,379.62,141.00,0.00),v40,z0,tPen\WObj:=wPaper;
    MoveL Offs(pOrigin,380.26,141.43,0.00),v40,z0,tPen\WObj:=wPaper;
    MoveL Offs(pOrigin,380.90,142.06,0.00),v40,z0,tPen\WObj:=wPaper;
    MoveL Offs(pOrigin,380.26,141.43,0.00),v40,z0,tPen\WObj:=wPaper;
    MoveL Offs(pOrigin,379.59,141.86,0.00),v40,z0,tPen\WObj:=wPaper;
    MoveL Offs(pOrigin,381.54,139.91,0.00),v40,z0,tPen\WObj:=wPaper;
    MoveL Offs(pOrigin,382.44,140.50,0.00),v40,z0,tPen\WObj:=wPaper;
    MoveL Offs(pOrigin,380.34,142.61,0.00),v40,z0,tPen\WObj:=wPaper;
    MoveL Offs(pOrigin,381.23,143.20,0.00),v40,z0,tPen\WObj:=wPaper;
    MoveL Offs(pOrigin,383.34,141.10,0.00),v40,z0,tPen\WObj:=wPaper;
    MoveL Offs(pOrigin,384.23,141.69,0.00),v40,z0,tPen\WObj:=wPaper;
    MoveL Offs(pOrigin,381.98,143.95,0.00),v40,z0,tPen\WObj:=wPaper;
    MoveL Offs(pOrigin,381.96,142.91,0.00),v40,z0,tPen\WObj:=wPaper;
    MoveL Offs(pOrigin,384.09,144.82,0.00),v40,z0,tPen\WObj:=wPaper;
    MoveL Offs(pOrigin,381.96,142.91,0.00),v40,z0,tPen\WObj:=wPaper;
    MoveL Offs(pOrigin,382.60,142.78,0.00),v40,z0,tPen\WObj:=wPaper;
    MoveL Offs(pOrigin,383.88,142.78,0.00),v40,z0,tPen\WObj:=wPaper;
    MoveL Offs(pOrigin,384.18,142.54,0.00),v40,z0,tPen\WObj:=wPaper;
    MoveL Offs(pOrigin,387.19,145.55,0.00),v40,z0,tPen\WObj:=wPaper;
    MoveL Offs(pOrigin,387.67,145.73,0.00),v40,z0,tPen\WObj:=wPaper;
    MoveL Offs(pOrigin,384.36,149.03,0.00),v40,z0,tPen\WObj:=wPaper;
    MoveL Offs(pOrigin,384.95,149.29,0.00),v40,z0,tPen\WObj:=wPaper;
    MoveL Offs(pOrigin,386.76,151.09,0.00),v40,z0,tPen\WObj:=wPaper;
    MoveL Offs(pOrigin,386.21,151.22,0.00),v40,z0,tPen\WObj:=wPaper;
    MoveL Offs(pOrigin,384.94,151.22,0.00),v40,z0,tPen\WObj:=wPaper;
    MoveL Offs(pOrigin,383.76,151.13,0.00),v40,z0,tPen\WObj:=wPaper;
    MoveL Offs(pOrigin,387.81,147.08,0.00),v40,z0,tPen\WObj:=wPaper;
    MoveL Offs(pOrigin,387.34,147.20,0.00),v40,z0,tPen\WObj:=wPaper;
    MoveL Offs(pOrigin,378.93,138.78,0.00),v40,z0,tPen\WObj:=wPaper;
    MoveL Offs(pOrigin,379.00,137.97,0.00),v40,z0,tPen\WObj:=wPaper;
    MoveL Offs(pOrigin,377.20,139.77,0.00),v40,z0,tPen\WObj:=wPaper;
    MoveL Offs(pOrigin,378.10,140.37,0.00),v40,z0,tPen\WObj:=wPaper;
    MoveL Offs(pOrigin,379.75,138.71,0.00),v40,fine,tPen\WObj:=wPaper;
    MoveL Offs(pOrigin,379.75,138.71,6.00),v60,z5,tPen\WObj:=wPaper;
    MoveL Offs(pOrigin,377.92,138.66,6.00),vTravel,z5,tPen\WObj:=wPaper;
    MoveL Offs(pOrigin,377.92,138.66,0.00),v60,z0,tPen\WObj:=wPaper;
    MoveL Offs(pOrigin,375.80,137.18,0.00),v40,z0,tPen\WObj:=wPaper;
    MoveL Offs(pOrigin,372.61,134.20,0.00),v40,fine,tPen\WObj:=wPaper;
    MoveL Offs(pOrigin,372.61,134.20,6.00),v60,z5,tPen\WObj:=wPaper;
    MoveL Offs(pOrigin,373.47,136.04,6.00),vTravel,z5,tPen\WObj:=wPaper;
    MoveL Offs(pOrigin,373.47,136.04,0.00),v60,z0,tPen\WObj:=wPaper;
    MoveL Offs(pOrigin,374.67,134.83,0.00),v40,fine,tPen\WObj:=wPaper;
    MoveL Offs(pOrigin,374.67,134.83,6.00),v60,z5,tPen\WObj:=wPaper;
    MoveL Offs(pOrigin,374.95,133.35,6.00),vTravel,z5,tPen\WObj:=wPaper;
    MoveL Offs(pOrigin,374.95,133.35,0.00),v60,z0,tPen\WObj:=wPaper;
    MoveL Offs(pOrigin,377.08,134.70,0.00),v40,z0,tPen\WObj:=wPaper;
    MoveL Offs(pOrigin,381.11,136.54,0.00),v40,z0,tPen\WObj:=wPaper;
    MoveL Offs(pOrigin,384.09,137.39,0.00),v40,z0,tPen\WObj:=wPaper;
    MoveL Offs(pOrigin,387.06,137.39,0.00),v40,z0,tPen\WObj:=wPaper;
    MoveL Offs(pOrigin,387.84,138.09,0.00),v40,z0,tPen\WObj:=wPaper;
    MoveL Offs(pOrigin,394.90,131.03,0.00),v40,fine,tPen\WObj:=wPaper;
    MoveL Offs(pOrigin,394.90,131.03,6.00),v60,z5,tPen\WObj:=wPaper;
    MoveL Offs(pOrigin,393.65,132.22,6.00),vTravel,z5,tPen\WObj:=wPaper;
    MoveL Offs(pOrigin,393.65,132.22,0.00),v60,z0,tPen\WObj:=wPaper;
    MoveL Offs(pOrigin,392.59,132.22,0.00),v40,fine,tPen\WObj:=wPaper;
    MoveL Offs(pOrigin,392.59,132.22,6.00),v60,z5,tPen\WObj:=wPaper;
    MoveL Offs(pOrigin,390.89,131.16,6.00),vTravel,z5,tPen\WObj:=wPaper;
    MoveL Offs(pOrigin,390.89,131.16,0.00),v60,z0,tPen\WObj:=wPaper;
    MoveL Offs(pOrigin,389.61,131.16,0.00),v40,z0,tPen\WObj:=wPaper;
    MoveL Offs(pOrigin,389.09,131.02,0.00),v40,z0,tPen\WObj:=wPaper;
    MoveL Offs(pOrigin,393.90,135.83,0.00),v40,z0,tPen\WObj:=wPaper;
    MoveL Offs(pOrigin,394.14,136.27,0.00),v40,z0,tPen\WObj:=wPaper;
    MoveL Offs(pOrigin,384.22,146.19,0.00),v40,z0,tPen\WObj:=wPaper;
    MoveL Offs(pOrigin,384.51,145.46,0.00),v40,z0,tPen\WObj:=wPaper;
    MoveL Offs(pOrigin,384.94,145.89,0.00),v40,z0,tPen\WObj:=wPaper;
    MoveL Offs(pOrigin,384.51,145.46,0.00),v40,z0,tPen\WObj:=wPaper;
    MoveL Offs(pOrigin,384.51,144.89,0.00),v40,z0,tPen\WObj:=wPaper;
    MoveL Offs(pOrigin,386.64,144.89,0.00),v40,z0,tPen\WObj:=wPaper;
    MoveL Offs(pOrigin,387.33,144.20,0.00),v40,z0,tPen\WObj:=wPaper;
    MoveL Offs(pOrigin,385.53,142.40,0.00),v40,z0,tPen\WObj:=wPaper;
    MoveL Offs(pOrigin,385.79,142.78,0.00),v40,z0,tPen\WObj:=wPaper;
    MoveL Offs(pOrigin,387.70,142.78,0.00),v40,z0,tPen\WObj:=wPaper;
    MoveL Offs(pOrigin,388.12,142.70,0.00),v40,z0,tPen\WObj:=wPaper;
    MoveL Offs(pOrigin,387.91,143.12,0.00),v40,z0,tPen\WObj:=wPaper;
    MoveL Offs(pOrigin,388.12,142.70,0.00),v40,z0,tPen\WObj:=wPaper;
    MoveL Offs(pOrigin,388.55,142.49,0.00),v40,z0,tPen\WObj:=wPaper;
    MoveL Offs(pOrigin,388.76,142.06,0.00),v40,z0,tPen\WObj:=wPaper;
    MoveL Offs(pOrigin,388.55,142.49,0.00),v40,z0,tPen\WObj:=wPaper;
    MoveL Offs(pOrigin,388.83,142.71,0.00),v40,z0,tPen\WObj:=wPaper;
    MoveL Offs(pOrigin,387.17,141.05,0.00),v40,z0,tPen\WObj:=wPaper;
    MoveL Offs(pOrigin,387.06,141.72,0.00),v40,z0,tPen\WObj:=wPaper;
    MoveL Offs(pOrigin,388.76,141.72,0.00),v40,z0,tPen\WObj:=wPaper;
    MoveL Offs(pOrigin,389.42,141.81,0.00),v40,z0,tPen\WObj:=wPaper;
    MoveL Offs(pOrigin,387.92,140.31,0.00),v40,z0,tPen\WObj:=wPaper;
    MoveL Offs(pOrigin,388.27,140.15,0.00),v40,z0,tPen\WObj:=wPaper;
    MoveL Offs(pOrigin,385.79,142.70,0.00),v40,z0,tPen\WObj:=wPaper;
    MoveL Offs(pOrigin,388.27,140.15,0.00),v40,z0,tPen\WObj:=wPaper;
    MoveL Offs(pOrigin,388.12,140.66,0.00),v40,z0,tPen\WObj:=wPaper;
    MoveL Offs(pOrigin,389.61,140.66,0.00),v40,z0,tPen\WObj:=wPaper;
    MoveL Offs(pOrigin,389.61,141.00,0.00),v40,z0,tPen\WObj:=wPaper;
    MoveL Offs(pOrigin,389.40,141.43,0.00),v40,z0,tPen\WObj:=wPaper;
    MoveL Offs(pOrigin,389.61,141.00,0.00),v40,z0,tPen\WObj:=wPaper;
    MoveL Offs(pOrigin,390.17,141.06,0.00),v40,z0,tPen\WObj:=wPaper;
    MoveL Offs(pOrigin,388.22,139.11,0.00),v40,z0,tPen\WObj:=wPaper;
    MoveL Offs(pOrigin,388.76,139.61,0.00),v40,z0,tPen\WObj:=wPaper;
    MoveL Offs(pOrigin,390.04,139.61,0.00),v40,z0,tPen\WObj:=wPaper;
    MoveL Offs(pOrigin,390.46,138.55,0.00),v40,z0,tPen\WObj:=wPaper;
    MoveL Offs(pOrigin,389.19,138.55,0.00),v40,fine,tPen\WObj:=wPaper;
    MoveL Offs(pOrigin,389.19,138.55,6.00),v60,z5,tPen\WObj:=wPaper;
    MoveL Offs(pOrigin,386.35,136.59,6.00),vTravel,z5,tPen\WObj:=wPaper;
    MoveL Offs(pOrigin,386.35,136.59,0.00),v60,z0,tPen\WObj:=wPaper;
    MoveL Offs(pOrigin,384.69,138.25,0.00),v40,fine,tPen\WObj:=wPaper;
    MoveL Offs(pOrigin,384.69,138.25,6.00),v60,z5,tPen\WObj:=wPaper;
    MoveL Offs(pOrigin,386.43,141.80,6.00),vTravel,z5,tPen\WObj:=wPaper;
    MoveL Offs(pOrigin,386.43,141.80,0.00),v60,z0,tPen\WObj:=wPaper;
    MoveL Offs(pOrigin,387.93,143.30,0.00),v40,z0,tPen\WObj:=wPaper;
    MoveL Offs(pOrigin,387.49,143.34,0.00),v40,z0,tPen\WObj:=wPaper;
    MoveL Offs(pOrigin,387.27,143.76,0.00),v40,z0,tPen\WObj:=wPaper;
    MoveL Offs(pOrigin,387.49,143.34,0.00),v40,z0,tPen\WObj:=wPaper;
    MoveL Offs(pOrigin,387.06,143.83,0.00),v40,z0,tPen\WObj:=wPaper;
    MoveL Offs(pOrigin,383.66,143.83,0.00),v40,z0,tPen\WObj:=wPaper;
    MoveL Offs(pOrigin,382.88,144.54,0.00),v40,z0,tPen\WObj:=wPaper;
    MoveL Offs(pOrigin,394.60,132.82,0.00),v40,fine,tPen\WObj:=wPaper;
    MoveL Offs(pOrigin,394.60,132.82,6.00),v60,z5,tPen\WObj:=wPaper;
  ENDPROC

  PROC DrawPart207()
    MoveL Offs(pOrigin,394.44,134.47,6.00),vTravel,z5,tPen\WObj:=wPaper;
    MoveL Offs(pOrigin,394.44,134.47,0.00),v60,z0,tPen\WObj:=wPaper;
    MoveL Offs(pOrigin,383.47,145.44,0.00),v40,fine,tPen\WObj:=wPaper;
    MoveL Offs(pOrigin,383.47,145.44,6.00),v60,z5,tPen\WObj:=wPaper;
    MoveL Offs(pOrigin,385.15,145.94,6.00),vTravel,z5,tPen\WObj:=wPaper;
    MoveL Offs(pOrigin,385.15,145.94,0.00),v60,z0,tPen\WObj:=wPaper;
    MoveL Offs(pOrigin,386.85,145.94,0.00),v40,z0,tPen\WObj:=wPaper;
    MoveL Offs(pOrigin,386.85,147.00,0.00),v40,z0,tPen\WObj:=wPaper;
    MoveL Offs(pOrigin,385.58,147.00,0.00),v40,z0,tPen\WObj:=wPaper;
    MoveL Offs(pOrigin,385.79,148.06,0.00),v40,z0,tPen\WObj:=wPaper;
    MoveL Offs(pOrigin,386.85,148.06,0.00),v40,z0,tPen\WObj:=wPaper;
    MoveL Offs(pOrigin,386.85,149.11,0.00),v40,z0,tPen\WObj:=wPaper;
    MoveL Offs(pOrigin,385.58,149.11,0.00),v40,fine,tPen\WObj:=wPaper;
    MoveL Offs(pOrigin,385.58,149.11,6.00),v60,z5,tPen\WObj:=wPaper;
    MoveL Offs(pOrigin,387.65,150.22,6.00),vTravel,z5,tPen\WObj:=wPaper;
    MoveL Offs(pOrigin,387.65,150.22,0.00),v60,z0,tPen\WObj:=wPaper;
    MoveL Offs(pOrigin,380.89,156.98,0.00),v40,fine,tPen\WObj:=wPaper;
    MoveL Offs(pOrigin,380.89,156.98,6.00),v60,z5,tPen\WObj:=wPaper;
    MoveL Offs(pOrigin,379.84,159.53,6.00),vTravel,z5,tPen\WObj:=wPaper;
    MoveL Offs(pOrigin,379.84,159.53,0.00),v60,z0,tPen\WObj:=wPaper;
    MoveL Offs(pOrigin,386.75,152.62,0.00),v40,fine,tPen\WObj:=wPaper;
    MoveL Offs(pOrigin,386.75,152.62,6.00),v60,z5,tPen\WObj:=wPaper;
    MoveL Offs(pOrigin,389.29,153.06,6.00),vTravel,z5,tPen\WObj:=wPaper;
    MoveL Offs(pOrigin,389.29,153.06,0.00),v60,z0,tPen\WObj:=wPaper;
    MoveL Offs(pOrigin,392.75,149.61,0.00),v40,z0,tPen\WObj:=wPaper;
    MoveL Offs(pOrigin,392.44,149.31,0.00),v40,z0,tPen\WObj:=wPaper;
    MoveL Offs(pOrigin,390.64,147.51,0.00),v40,z0,tPen\WObj:=wPaper;
    MoveL Offs(pOrigin,391.10,147.00,0.00),v40,z0,tPen\WObj:=wPaper;
    MoveL Offs(pOrigin,392.16,147.00,0.00),v40,fine,tPen\WObj:=wPaper;
    MoveL Offs(pOrigin,392.16,147.00,6.00),v60,z5,tPen\WObj:=wPaper;
    MoveL Offs(pOrigin,391.95,149.11,6.00),vTravel,z5,tPen\WObj:=wPaper;
    MoveL Offs(pOrigin,391.95,149.11,0.00),v60,z0,tPen\WObj:=wPaper;
    MoveL Offs(pOrigin,390.89,149.11,0.00),v40,z0,tPen\WObj:=wPaper;
    MoveL Offs(pOrigin,390.34,148.70,0.00),v40,z0,tPen\WObj:=wPaper;
    MoveL Offs(pOrigin,392.30,150.66,0.00),v40,z0,tPen\WObj:=wPaper;
    MoveL Offs(pOrigin,392.89,150.96,0.00),v40,z0,tPen\WObj:=wPaper;
    MoveL Offs(pOrigin,389.44,154.41,0.00),v40,z0,tPen\WObj:=wPaper;
    MoveL Offs(pOrigin,389.91,154.25,0.00),v40,z0,tPen\WObj:=wPaper;
    MoveL Offs(pOrigin,391.56,155.90,0.00),v40,z0,tPen\WObj:=wPaper;
    MoveL Offs(pOrigin,391.31,155.45,0.00),v40,z0,tPen\WObj:=wPaper;
    MoveL Offs(pOrigin,390.25,155.45,0.00),v40,z0,tPen\WObj:=wPaper;
    MoveL Offs(pOrigin,389.62,155.44,0.00),v40,z0,tPen\WObj:=wPaper;
    MoveL Offs(pOrigin,391.42,157.25,0.00),v40,z0,tPen\WObj:=wPaper;
    MoveL Offs(pOrigin,391.10,157.56,0.00),v40,z0,tPen\WObj:=wPaper;
    MoveL Offs(pOrigin,390.04,157.56,0.00),v40,fine,tPen\WObj:=wPaper;
    MoveL Offs(pOrigin,390.04,157.56,6.00),v60,z5,tPen\WObj:=wPaper;
    MoveL Offs(pOrigin,392.12,157.70,6.00),vTravel,z5,tPen\WObj:=wPaper;
    MoveL Offs(pOrigin,392.12,157.70,0.00),v60,z0,tPen\WObj:=wPaper;
    MoveL Offs(pOrigin,388.67,161.15,0.00),v40,z0,tPen\WObj:=wPaper;
    MoveL Offs(pOrigin,389.33,161.13,0.00),v40,z0,tPen\WObj:=wPaper;
    MoveL Offs(pOrigin,390.99,162.79,0.00),v40,z0,tPen\WObj:=wPaper;
    MoveL Offs(pOrigin,390.67,162.84,0.00),v40,z0,tPen\WObj:=wPaper;
    MoveL Offs(pOrigin,389.61,162.84,0.00),v40,z0,tPen\WObj:=wPaper;
    MoveL Offs(pOrigin,388.89,163.68,0.00),v40,z0,tPen\WObj:=wPaper;
    MoveL Offs(pOrigin,390.84,165.63,0.00),v40,z0,tPen\WObj:=wPaper;
    MoveL Offs(pOrigin,391.35,165.94,0.00),v40,z0,tPen\WObj:=wPaper;
    MoveL Offs(pOrigin,387.89,169.40,0.00),v40,z0,tPen\WObj:=wPaper;
    MoveL Offs(pOrigin,388.16,170.42,0.00),v40,z0,tPen\WObj:=wPaper;
    MoveL Offs(pOrigin,390.27,172.52,0.00),v40,z0,tPen\WObj:=wPaper;
    MoveL Offs(pOrigin,390.58,172.68,0.00),v40,z0,tPen\WObj:=wPaper;
    MoveL Offs(pOrigin,387.12,176.14,0.00),v40,fine,tPen\WObj:=wPaper;
    MoveL Offs(pOrigin,387.12,176.14,6.00),v60,z5,tPen\WObj:=wPaper;
    MoveL Offs(pOrigin,387.58,177.31,6.00),vTravel,z5,tPen\WObj:=wPaper;
    MoveL Offs(pOrigin,387.58,177.31,0.00),v60,z0,tPen\WObj:=wPaper;
    MoveL Offs(pOrigin,389.39,179.11,0.00),v40,z0,tPen\WObj:=wPaper;
    MoveL Offs(pOrigin,389.96,179.28,0.00),v40,z0,tPen\WObj:=wPaper;
    MoveL Offs(pOrigin,386.51,182.73,0.00),v40,z0,tPen\WObj:=wPaper;
    MoveL Offs(pOrigin,387.15,182.85,0.00),v40,z0,tPen\WObj:=wPaper;
    MoveL Offs(pOrigin,388.96,184.65,0.00),v40,fine,tPen\WObj:=wPaper;
    MoveL Offs(pOrigin,388.96,184.65,6.00),v60,z5,tPen\WObj:=wPaper;
    MoveL Offs(pOrigin,389.34,185.87,6.00),vTravel,z5,tPen\WObj:=wPaper;
    MoveL Offs(pOrigin,389.34,185.87,0.00),v60,z0,tPen\WObj:=wPaper;
    MoveL Offs(pOrigin,386.04,189.18,0.00),v40,z0,tPen\WObj:=wPaper;
    MoveL Offs(pOrigin,386.57,189.74,0.00),v40,z0,tPen\WObj:=wPaper;
    MoveL Offs(pOrigin,388.38,191.54,0.00),v40,fine,tPen\WObj:=wPaper;
    MoveL Offs(pOrigin,388.38,191.54,6.00),v60,z5,tPen\WObj:=wPaper;
    MoveL Offs(pOrigin,386.43,192.58,6.00),vTravel,z5,tPen\WObj:=wPaper;
    MoveL Offs(pOrigin,386.43,192.58,0.00),v60,z0,tPen\WObj:=wPaper;
    MoveL Offs(pOrigin,388.09,194.24,0.00),v40,z0,tPen\WObj:=wPaper;
    MoveL Offs(pOrigin,388.72,193.96,0.00),v40,z0,tPen\WObj:=wPaper;
    MoveL Offs(pOrigin,385.26,197.42,0.00),v40,z0,tPen\WObj:=wPaper;
    MoveL Offs(pOrigin,385.85,197.97,0.00),v40,z0,tPen\WObj:=wPaper;
    MoveL Offs(pOrigin,387.65,199.78,0.00),v40,z0,tPen\WObj:=wPaper;
    MoveL Offs(pOrigin,387.95,199.21,0.00),v40,z0,tPen\WObj:=wPaper;
    MoveL Offs(pOrigin,384.80,202.36,0.00),v40,z0,tPen\WObj:=wPaper;
    MoveL Offs(pOrigin,385.41,202.02,0.00),v40,z0,tPen\WObj:=wPaper;
    MoveL Offs(pOrigin,387.22,203.82,0.00),v40,z0,tPen\WObj:=wPaper;
    MoveL Offs(pOrigin,387.79,203.85,0.00),v40,z0,tPen\WObj:=wPaper;
    MoveL Offs(pOrigin,384.33,207.31,0.00),v40,z0,tPen\WObj:=wPaper;
    MoveL Offs(pOrigin,384.98,207.56,0.00),v40,z0,tPen\WObj:=wPaper;
    MoveL Offs(pOrigin,386.78,209.36,0.00),v40,z0,tPen\WObj:=wPaper;
    MoveL Offs(pOrigin,386.42,209.30,0.00),v40,z0,tPen\WObj:=wPaper;
    MoveL Offs(pOrigin,385.36,209.30,0.00),v40,fine,tPen\WObj:=wPaper;
    MoveL Offs(pOrigin,385.36,209.30,6.00),v60,z5,tPen\WObj:=wPaper;
    MoveL Offs(pOrigin,386.93,208.01,6.00),vTravel,z5,tPen\WObj:=wPaper;
    MoveL Offs(pOrigin,386.93,208.01,0.00),v60,z0,tPen\WObj:=wPaper;
    MoveL Offs(pOrigin,385.28,206.36,0.00),v40,fine,tPen\WObj:=wPaper;
    MoveL Offs(pOrigin,385.28,206.36,6.00),v60,z5,tPen\WObj:=wPaper;
    MoveL Offs(pOrigin,382.24,206.41,6.00),vTravel,z5,tPen\WObj:=wPaper;
    MoveL Offs(pOrigin,382.24,206.41,0.00),v60,z0,tPen\WObj:=wPaper;
    MoveL Offs(pOrigin,379.38,209.27,0.00),v40,z0,tPen\WObj:=wPaper;
    MoveL Offs(pOrigin,380.19,208.74,0.00),v40,z0,tPen\WObj:=wPaper;
    MoveL Offs(pOrigin,381.84,210.40,0.00),v40,z0,tPen\WObj:=wPaper;
    MoveL Offs(pOrigin,382.53,210.61,0.00),v40,z0,tPen\WObj:=wPaper;
    MoveL Offs(pOrigin,379.82,213.31,0.00),v40,z0,tPen\WObj:=wPaper;
    MoveL Offs(pOrigin,380.36,213.39,0.00),v40,z0,tPen\WObj:=wPaper;
    MoveL Offs(pOrigin,381.86,214.89,0.00),v40,z0,tPen\WObj:=wPaper;
    MoveL Offs(pOrigin,382.66,214.95,0.00),v40,z0,tPen\WObj:=wPaper;
    MoveL Offs(pOrigin,379.51,218.11,0.00),v40,z0,tPen\WObj:=wPaper;
    MoveL Offs(pOrigin,380.22,217.73,0.00),v40,z0,tPen\WObj:=wPaper;
    MoveL Offs(pOrigin,381.72,219.23,0.00),v40,z0,tPen\WObj:=wPaper;
    MoveL Offs(pOrigin,382.35,218.25,0.00),v40,z0,tPen\WObj:=wPaper;
    MoveL Offs(pOrigin,379.35,221.25,0.00),v40,z0,tPen\WObj:=wPaper;
    MoveL Offs(pOrigin,379.93,221.92,0.00),v40,z0,tPen\WObj:=wPaper;
    MoveL Offs(pOrigin,381.59,223.58,0.00),v40,fine,tPen\WObj:=wPaper;
    MoveL Offs(pOrigin,381.59,223.58,6.00),v60,z5,tPen\WObj:=wPaper;
    MoveL Offs(pOrigin,382.93,223.43,6.00),vTravel,z5,tPen\WObj:=wPaper;
    MoveL Offs(pOrigin,382.93,223.43,0.00),v60,z0,tPen\WObj:=wPaper;
    MoveL Offs(pOrigin,384.44,224.93,0.00),v40,z0,tPen\WObj:=wPaper;
    MoveL Offs(pOrigin,385.18,224.38,0.00),v40,z0,tPen\WObj:=wPaper;
  ENDPROC

  PROC DrawPart208()
    MoveL Offs(pOrigin,374.81,234.75,0.00),v40,fine,tPen\WObj:=wPaper;
    MoveL Offs(pOrigin,374.81,234.75,6.00),v60,z5,tPen\WObj:=wPaper;
    MoveL Offs(pOrigin,374.73,236.14,6.00),vTravel,z5,tPen\WObj:=wPaper;
    MoveL Offs(pOrigin,374.73,236.14,0.00),v60,z0,tPen\WObj:=wPaper;
    MoveL Offs(pOrigin,376.39,237.79,0.00),v40,fine,tPen\WObj:=wPaper;
    MoveL Offs(pOrigin,376.39,237.79,6.00),v60,z5,tPen\WObj:=wPaper;
    MoveL Offs(pOrigin,375.16,236.20,6.00),vTravel,z5,tPen\WObj:=wPaper;
    MoveL Offs(pOrigin,375.16,236.20,0.00),v60,z0,tPen\WObj:=wPaper;
    MoveL Offs(pOrigin,375.38,235.77,0.00),v40,z0,tPen\WObj:=wPaper;
    MoveL Offs(pOrigin,375.16,236.20,0.00),v40,fine,tPen\WObj:=wPaper;
    MoveL Offs(pOrigin,375.16,236.20,6.00),v60,z5,tPen\WObj:=wPaper;
    MoveL Offs(pOrigin,376.23,234.65,6.00),vTravel,z5,tPen\WObj:=wPaper;
    MoveL Offs(pOrigin,376.23,234.65,0.00),v60,z0,tPen\WObj:=wPaper;
    MoveL Offs(pOrigin,378.03,236.45,0.00),v40,fine,tPen\WObj:=wPaper;
    MoveL Offs(pOrigin,378.03,236.45,6.00),v60,z5,tPen\WObj:=wPaper;
    MoveL Offs(pOrigin,379.20,235.14,6.00),vTravel,z5,tPen\WObj:=wPaper;
    MoveL Offs(pOrigin,379.20,235.14,0.00),v60,z0,tPen\WObj:=wPaper;
    MoveL Offs(pOrigin,377.71,236.62,0.00),v40,z0,tPen\WObj:=wPaper;
    MoveL Offs(pOrigin,379.20,235.14,0.00),v40,fine,tPen\WObj:=wPaper;
    MoveL Offs(pOrigin,379.20,235.14,6.00),v60,z5,tPen\WObj:=wPaper;
    MoveL Offs(pOrigin,380.48,230.46,6.00),vTravel,z5,tPen\WObj:=wPaper;
    MoveL Offs(pOrigin,380.48,230.46,0.00),v60,z0,tPen\WObj:=wPaper;
    MoveL Offs(pOrigin,380.26,230.89,0.00),v40,z0,tPen\WObj:=wPaper;
    MoveL Offs(pOrigin,380.48,230.46,0.00),v40,z0,tPen\WObj:=wPaper;
    MoveL Offs(pOrigin,380.69,230.42,0.00),v40,z0,tPen\WObj:=wPaper;
    MoveL Offs(pOrigin,381.96,230.42,0.00),v40,z0,tPen\WObj:=wPaper;
    MoveL Offs(pOrigin,382.51,230.47,0.00),v40,z0,tPen\WObj:=wPaper;
    MoveL Offs(pOrigin,379.20,227.16,0.00),v40,z0,tPen\WObj:=wPaper;
    MoveL Offs(pOrigin,378.73,226.35,0.00),v40,z0,tPen\WObj:=wPaper;
    MoveL Offs(pOrigin,386.24,218.83,0.00),v40,z0,tPen\WObj:=wPaper;
    MoveL Offs(pOrigin,385.76,218.80,0.00),v40,z0,tPen\WObj:=wPaper;
    MoveL Offs(pOrigin,383.96,216.99,0.00),v40,z0,tPen\WObj:=wPaper;
    MoveL Offs(pOrigin,383.40,217.20,0.00),v40,z0,tPen\WObj:=wPaper;
    MoveL Offs(pOrigin,386.86,213.74,0.00),v40,z0,tPen\WObj:=wPaper;
    MoveL Offs(pOrigin,386.35,213.41,0.00),v40,z0,tPen\WObj:=wPaper;
    MoveL Offs(pOrigin,384.54,211.60,0.00),v40,z0,tPen\WObj:=wPaper;
    MoveL Offs(pOrigin,384.02,212.10,0.00),v40,z0,tPen\WObj:=wPaper;
    MoveL Offs(pOrigin,387.47,208.64,0.00),v40,fine,tPen\WObj:=wPaper;
    MoveL Offs(pOrigin,387.47,208.64,6.00),v60,z5,tPen\WObj:=wPaper;
    MoveL Offs(pOrigin,382.23,207.91,6.00),vTravel,z5,tPen\WObj:=wPaper;
    MoveL Offs(pOrigin,382.23,207.91,0.00),v60,z0,tPen\WObj:=wPaper;
    MoveL Offs(pOrigin,379.68,210.47,0.00),v40,z0,tPen\WObj:=wPaper;
    MoveL Offs(pOrigin,380.20,210.24,0.00),v40,z0,tPen\WObj:=wPaper;
    MoveL Offs(pOrigin,381.85,211.89,0.00),v40,z0,tPen\WObj:=wPaper;
    MoveL Offs(pOrigin,382.67,211.96,0.00),v40,z0,tPen\WObj:=wPaper;
    MoveL Offs(pOrigin,379.82,214.81,0.00),v40,z0,tPen\WObj:=wPaper;
    MoveL Offs(pOrigin,380.36,214.88,0.00),v40,z0,tPen\WObj:=wPaper;
    MoveL Offs(pOrigin,381.86,216.39,0.00),v40,z0,tPen\WObj:=wPaper;
    MoveL Offs(pOrigin,382.66,216.45,0.00),v40,z0,tPen\WObj:=wPaper;
    MoveL Offs(pOrigin,379.50,219.60,0.00),v40,z0,tPen\WObj:=wPaper;
    MoveL Offs(pOrigin,380.22,219.23,0.00),v40,z0,tPen\WObj:=wPaper;
    MoveL Offs(pOrigin,381.73,220.73,0.00),v40,fine,tPen\WObj:=wPaper;
    MoveL Offs(pOrigin,381.73,220.73,6.00),v60,z5,tPen\WObj:=wPaper;
    MoveL Offs(pOrigin,381.58,222.08,6.00),vTravel,z5,tPen\WObj:=wPaper;
    MoveL Offs(pOrigin,381.58,222.08,0.00),v60,z0,tPen\WObj:=wPaper;
    MoveL Offs(pOrigin,379.93,220.43,0.00),v40,fine,tPen\WObj:=wPaper;
    MoveL Offs(pOrigin,379.93,220.43,6.00),v60,z5,tPen\WObj:=wPaper;
    MoveL Offs(pOrigin,377.97,218.47,6.00),vTravel,z5,tPen\WObj:=wPaper;
    MoveL Offs(pOrigin,377.97,218.47,0.00),v60,z0,tPen\WObj:=wPaper;
    MoveL Offs(pOrigin,375.57,216.07,0.00),v40,z0,tPen\WObj:=wPaper;
    MoveL Offs(pOrigin,376.22,215.64,0.00),v40,z0,tPen\WObj:=wPaper;
    MoveL Offs(pOrigin,377.29,215.64,0.00),v40,fine,tPen\WObj:=wPaper;
    MoveL Offs(pOrigin,377.29,215.64,6.00),v60,z5,tPen\WObj:=wPaper;
    MoveL Offs(pOrigin,378.31,216.31,6.00),vTravel,z5,tPen\WObj:=wPaper;
    MoveL Offs(pOrigin,378.31,216.31,0.00),v60,z0,tPen\WObj:=wPaper;
    MoveL Offs(pOrigin,373.81,220.82,0.00),v40,fine,tPen\WObj:=wPaper;
    MoveL Offs(pOrigin,373.81,220.82,6.00),v60,z5,tPen\WObj:=wPaper;
    MoveL Offs(pOrigin,373.20,222.92,6.00),vTravel,z5,tPen\WObj:=wPaper;
    MoveL Offs(pOrigin,373.20,222.92,0.00),v60,z0,tPen\WObj:=wPaper;
    MoveL Offs(pOrigin,378.61,217.51,0.00),v40,fine,tPen\WObj:=wPaper;
    MoveL Offs(pOrigin,378.61,217.51,6.00),v60,z5,tPen\WObj:=wPaper;
    MoveL Offs(pOrigin,379.81,216.31,6.00),vTravel,z5,tPen\WObj:=wPaper;
    MoveL Offs(pOrigin,379.81,216.31,0.00),v60,z0,tPen\WObj:=wPaper;
    MoveL Offs(pOrigin,382.67,213.45,0.00),v40,z0,tPen\WObj:=wPaper;
    MoveL Offs(pOrigin,381.85,213.39,0.00),v40,z0,tPen\WObj:=wPaper;
    MoveL Offs(pOrigin,380.20,211.74,0.00),v40,z0,tPen\WObj:=wPaper;
    MoveL Offs(pOrigin,379.67,211.96,0.00),v40,z0,tPen\WObj:=wPaper;
    MoveL Offs(pOrigin,382.23,209.41,0.00),v40,z0,tPen\WObj:=wPaper;
    MoveL Offs(pOrigin,381.84,208.90,0.00),v40,z0,tPen\WObj:=wPaper;
    MoveL Offs(pOrigin,380.19,207.24,0.00),v40,z0,tPen\WObj:=wPaper;
    MoveL Offs(pOrigin,379.39,207.77,0.00),v40,z0,tPen\WObj:=wPaper;
    MoveL Offs(pOrigin,382.09,205.07,0.00),v40,z0,tPen\WObj:=wPaper;
    MoveL Offs(pOrigin,381.68,205.75,0.00),v40,z0,tPen\WObj:=wPaper;
    MoveL Offs(pOrigin,379.88,203.95,0.00),v40,z0,tPen\WObj:=wPaper;
    MoveL Offs(pOrigin,379.25,203.43,0.00),v40,z0,tPen\WObj:=wPaper;
    MoveL Offs(pOrigin,381.66,201.02,0.00),v40,z0,tPen\WObj:=wPaper;
    MoveL Offs(pOrigin,381.22,200.81,0.00),v40,z0,tPen\WObj:=wPaper;
    MoveL Offs(pOrigin,379.41,199.00,0.00),v40,z0,tPen\WObj:=wPaper;
    MoveL Offs(pOrigin,378.81,199.38,0.00),v40,z0,tPen\WObj:=wPaper;
    MoveL Offs(pOrigin,381.22,196.98,0.00),v40,z0,tPen\WObj:=wPaper;
    MoveL Offs(pOrigin,380.76,197.36,0.00),v40,z0,tPen\WObj:=wPaper;
    MoveL Offs(pOrigin,379.10,195.71,0.00),v40,z0,tPen\WObj:=wPaper;
    MoveL Offs(pOrigin,378.38,195.34,0.00),v40,z0,tPen\WObj:=wPaper;
    MoveL Offs(pOrigin,380.78,192.94,0.00),v40,z0,tPen\WObj:=wPaper;
    MoveL Offs(pOrigin,380.15,193.76,0.00),v40,z0,tPen\WObj:=wPaper;
    MoveL Offs(pOrigin,378.64,192.26,0.00),v40,z0,tPen\WObj:=wPaper;
    MoveL Offs(pOrigin,378.24,192.49,0.00),v40,z0,tPen\WObj:=wPaper;
    MoveL Offs(pOrigin,380.34,190.39,0.00),v40,fine,tPen\WObj:=wPaper;
    MoveL Offs(pOrigin,380.34,190.39,6.00),v60,z5,tPen\WObj:=wPaper;
    MoveL Offs(pOrigin,379.08,188.22,6.00),vTravel,z5,tPen\WObj:=wPaper;
    MoveL Offs(pOrigin,379.08,188.22,0.00),v60,z0,tPen\WObj:=wPaper;
    MoveL Offs(pOrigin,374.12,183.26,0.00),v40,fine,tPen\WObj:=wPaper;
    MoveL Offs(pOrigin,374.12,183.26,6.00),v60,z5,tPen\WObj:=wPaper;
    MoveL Offs(pOrigin,369.42,184.88,6.00),vTravel,z5,tPen\WObj:=wPaper;
    MoveL Offs(pOrigin,369.42,184.88,0.00),v60,z0,tPen\WObj:=wPaper;
    MoveL Offs(pOrigin,367.47,186.84,0.00),v40,z0,tPen\WObj:=wPaper;
    MoveL Offs(pOrigin,367.73,186.26,0.00),v40,z0,tPen\WObj:=wPaper;
    MoveL Offs(pOrigin,367.94,186.69,0.00),v40,z0,tPen\WObj:=wPaper;
    MoveL Offs(pOrigin,367.73,186.26,0.00),v40,z0,tPen\WObj:=wPaper;
    MoveL Offs(pOrigin,366.87,185.94,0.00),v40,z0,tPen\WObj:=wPaper;
    MoveL Offs(pOrigin,368.83,183.99,0.00),v40,fine,tPen\WObj:=wPaper;
    MoveL Offs(pOrigin,368.83,183.99,6.00),v60,z5,tPen\WObj:=wPaper;
    MoveL Offs(pOrigin,368.89,185.49,6.00),vTravel,z5,tPen\WObj:=wPaper;
    MoveL Offs(pOrigin,368.89,185.49,0.00),v60,z0,tPen\WObj:=wPaper;
    MoveL Offs(pOrigin,365.43,182.03,0.00),v40,z0,tPen\WObj:=wPaper;
    MoveL Offs(pOrigin,365.09,181.75,0.00),v40,z0,tPen\WObj:=wPaper;
    MoveL Offs(pOrigin,367.04,179.80,0.00),v40,z0,tPen\WObj:=wPaper;
    MoveL Offs(pOrigin,366.77,180.39,0.00),v40,z0,tPen\WObj:=wPaper;
    MoveL Offs(pOrigin,363.77,177.38,0.00),v40,z0,tPen\WObj:=wPaper;
    MoveL Offs(pOrigin,363.30,177.56,0.00),v40,z0,tPen\WObj:=wPaper;
  ENDPROC

